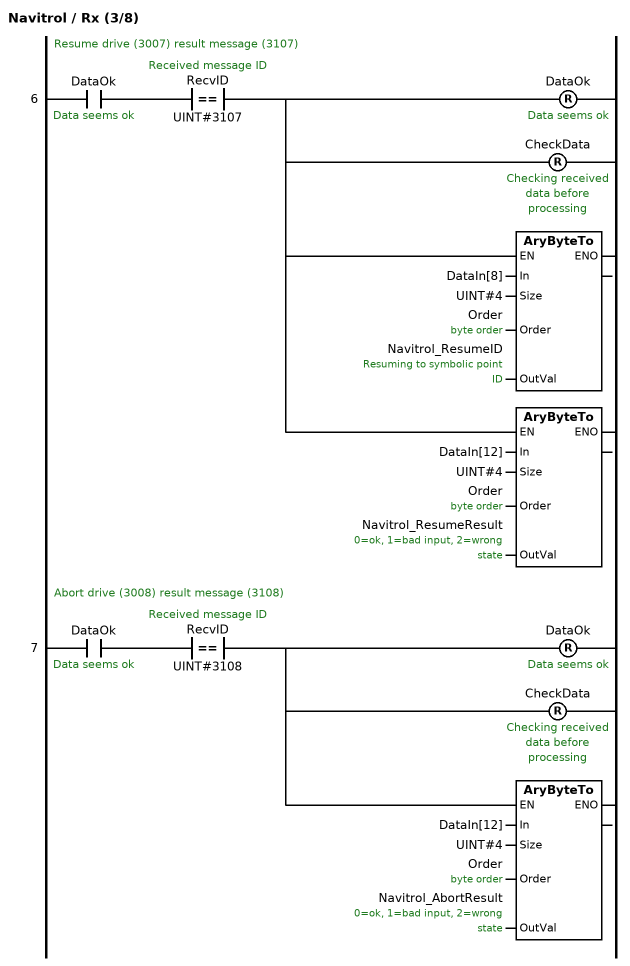
(* Rung 6: Resume drive (3007) result message (3107) *)
_p10 := DataOk AND (RecvID = UINT#3107);
IF _p10 THEN
    DataOk := FALSE;
    CheckData := FALSE;
    AryByteTo(In := DataIn[8], Size := UINT#4, Order := Order, OutVal := Navitrol_ResumeID);
    AryByteTo(In := DataIn[12], Size := UINT#4, Order := Order, OutVal := Navitrol_ResumeResult);
END_IF;
(* Rung 7: Abort drive (3008) result message (3108) *)
_p11 := DataOk AND (RecvID = UINT#3108);
IF _p11 THEN
    DataOk := FALSE;
    CheckData := FALSE;
    AryByteTo(In := DataIn[12], Size := UINT#4, Order := Order, OutVal := Navitrol_AbortResult);
END_IF;

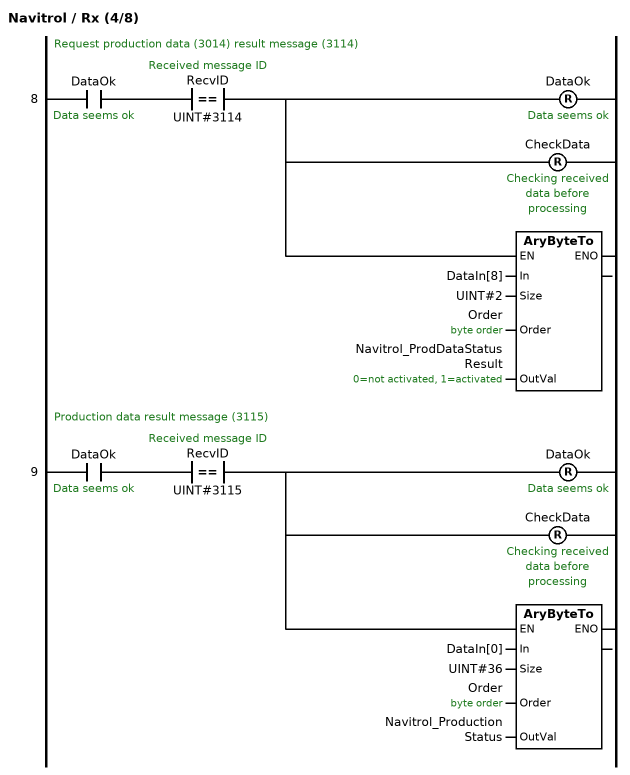
(* Rung 8: Request production data (3014) result message (3114) *)
_p12 := DataOk AND (RecvID = UINT#3114);
IF _p12 THEN
    DataOk := FALSE;
    CheckData := FALSE;
    AryByteTo(In := DataIn[8], Size := UINT#2, Order := Order, OutVal := Navitrol_ProdDataStatusResult);
END_IF;
(* Rung 9: Production data result message (3115) *)
_p13 := DataOk AND (RecvID = UINT#3115);
IF _p13 THEN
    DataOk := FALSE;
    CheckData := FALSE;
    AryByteTo(In := DataIn[0], Size := UINT#36, Order := Order, OutVal := Navitrol_ProductionStatus);
END_IF;

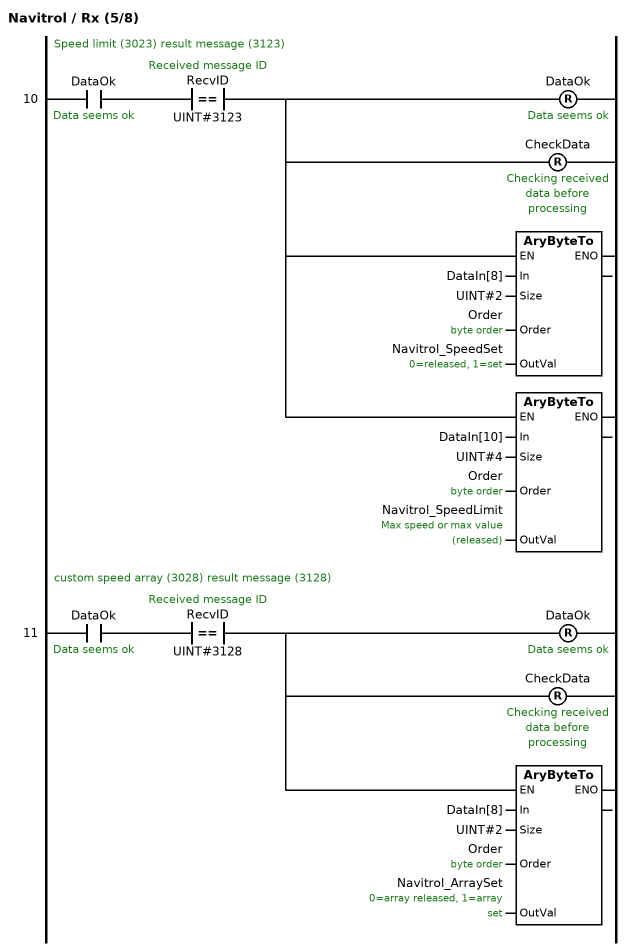
(* Rung 10: Speed limit (3023) result message (3123) *)
_p14 := DataOk AND (RecvID = UINT#3123);
IF _p14 THEN
    DataOk := FALSE;
    CheckData := FALSE;
    AryByteTo(In := DataIn[8], Size := UINT#2, Order := Order, OutVal := Navitrol_SpeedSet);
    AryByteTo(In := DataIn[10], Size := UINT#4, Order := Order, OutVal := Navitrol_SpeedLimit);
END_IF;
(* Rung 11: custom speed array (3028) result message (3128) *)
_p15 := DataOk AND (RecvID = UINT#3128);
IF _p15 THEN
    DataOk := FALSE;
    CheckData := FALSE;
    AryByteTo(In := DataIn[8], Size := UINT#2, Order := Order, OutVal := Navitrol_ArraySet);
END_IF;

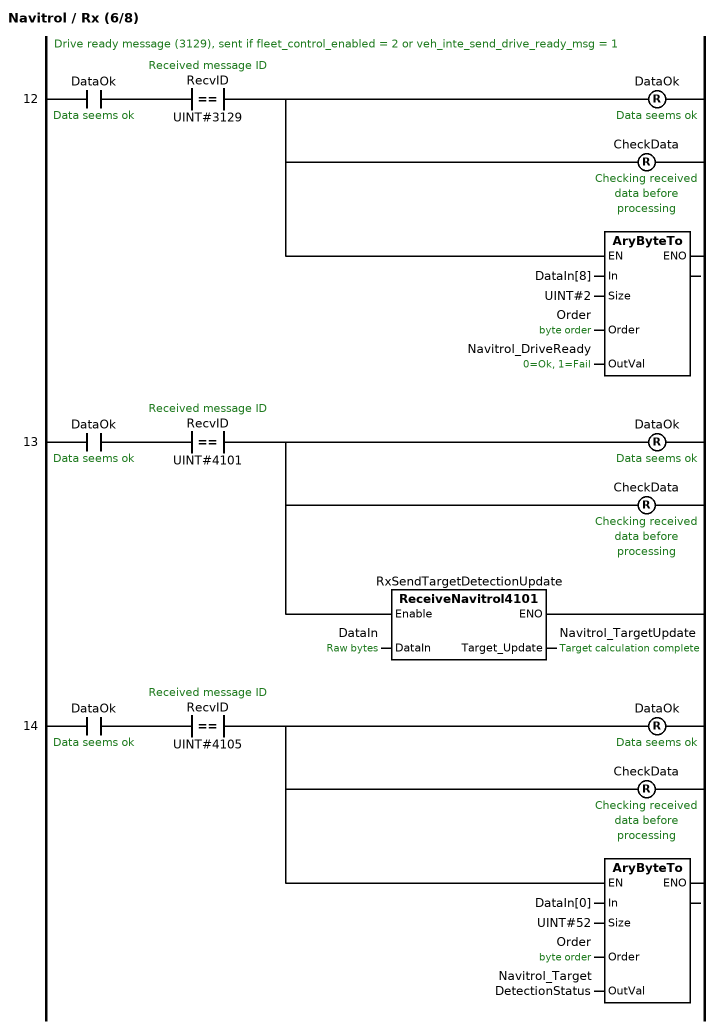
(* Rung 12: Drive ready message (3129), sent if fleet_control_enabled = 2 or veh_inte_send_drive_ready_msg = 1 *)
_p16 := DataOk AND (RecvID = UINT#3129);
IF _p16 THEN
    DataOk := FALSE;
    CheckData := FALSE;
    AryByteTo(In := DataIn[8], Size := UINT#2, Order := Order, OutVal := Navitrol_DriveReady);
END_IF;
(* Rung 13 *)
_p17 := DataOk AND (RecvID = UINT#4101);
IF _p17 THEN
    DataOk := FALSE;
    CheckData := FALSE;
END_IF;
RxSendTargetDetectionUpdate(Enable := _p17, DataIn := DataIn, Target_Update => Navitrol_TargetUpdate);
(* Rung 14 *)
_p18 := DataOk AND (RecvID = UINT#4105);
IF _p18 THEN
    DataOk := FALSE;
    CheckData := FALSE;
    AryByteTo(In := DataIn[0], Size := UINT#52, Order := Order, OutVal := Navitrol_TargetDetectionStatus);
END_IF;

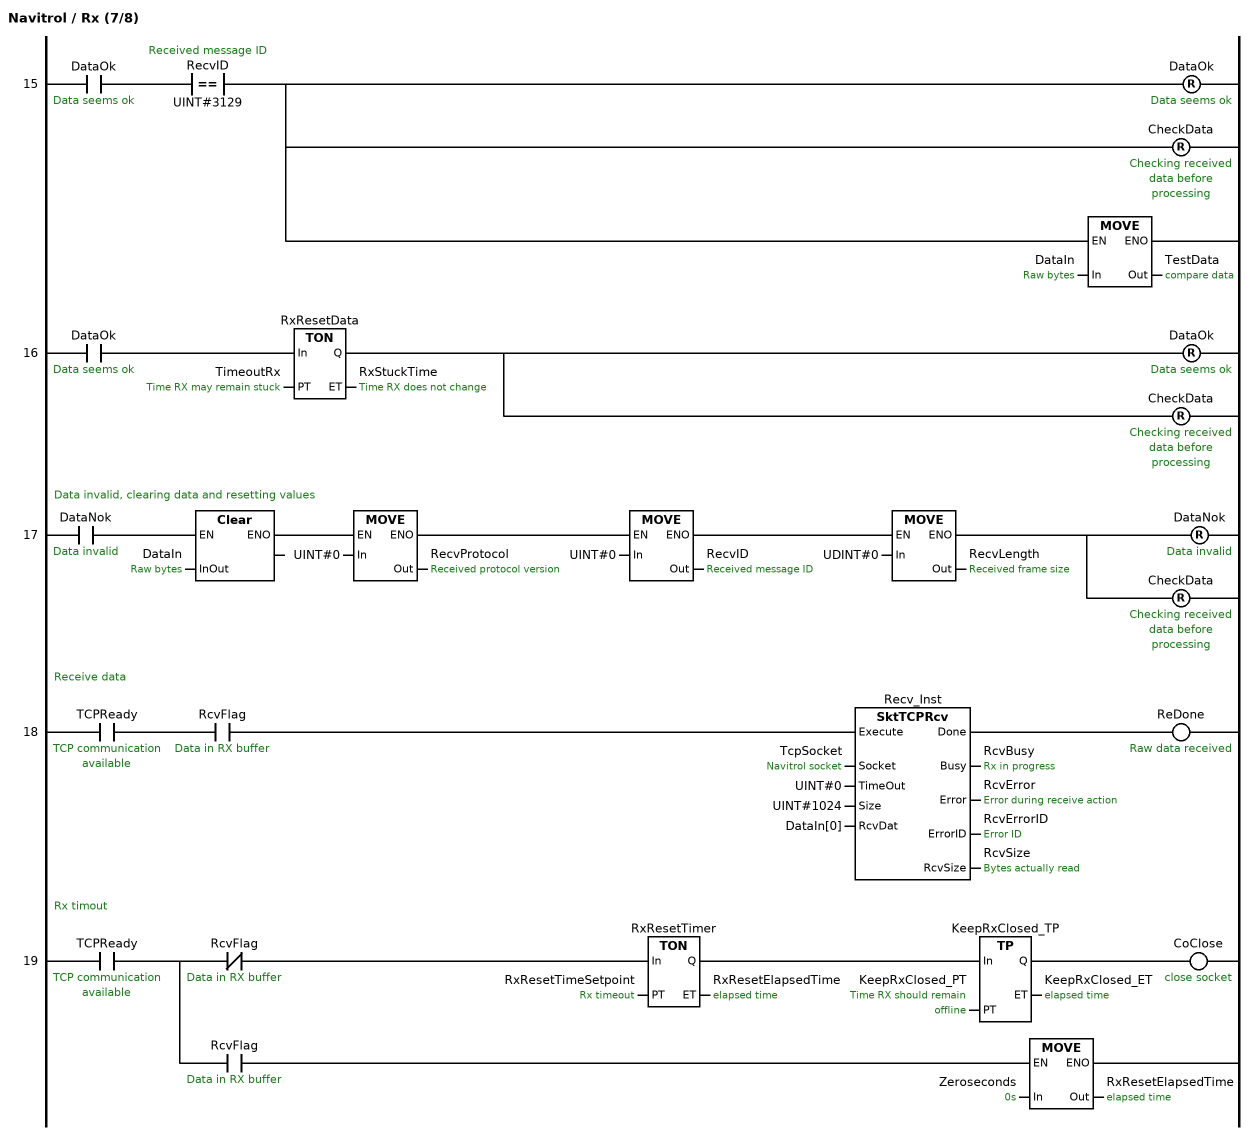
(* Rung 15 *)
_p19 := DataOk AND (RecvID = UINT#3129);
IF _p19 THEN
    DataOk := FALSE;
    CheckData := FALSE;
    TestData := DataIn;
END_IF;
(* Rung 16 *)
RxResetData(In := DataOk, PT := TimeoutRx, ET => RxStuckTime);
IF RxResetData.Q THEN
    DataOk := FALSE;
    CheckData := FALSE;
END_IF;
(* Rung 17: Data invalid, clearing data and resetting values *)
IF DataNok THEN
    Clear(InOut := DataIn);
    RecvProtocol := UINT#0;
    RecvID := UINT#0;
    RecvLength := UDINT#0;
END_IF;
_p20 := DataNok;
IF _p20 THEN
    DataNok := FALSE;
    CheckData := FALSE;
END_IF;
(* Rung 18: Receive data *)
Recv_Inst(Execute := TCPReady AND RcvFlag, Socket := TcpSocket, TimeOut := UINT#0, Size := UINT#1024, RcvDat := DataIn[0], Busy => RcvBusy, Error => RcvError, ErrorID => RcvErrorID, RcvSize => RcvSize);
ReDone := Recv_Inst.Done;
(* Rung 19: Rx timout *)
RxResetTimer(In := TCPReady AND NOT RcvFlag, PT := RxResetTimeSetpoint, ET => RxResetElapsedTime);
KeepRxClosed_TP(In := RxResetTimer.Q, PT := KeepRxClosed_PT, ET => KeepRxClosed_ET);
CoClose := KeepRxClosed_TP.Q;
IF TCPReady AND RcvFlag THEN RxResetElapsedTime := Zeroseconds; END_IF;

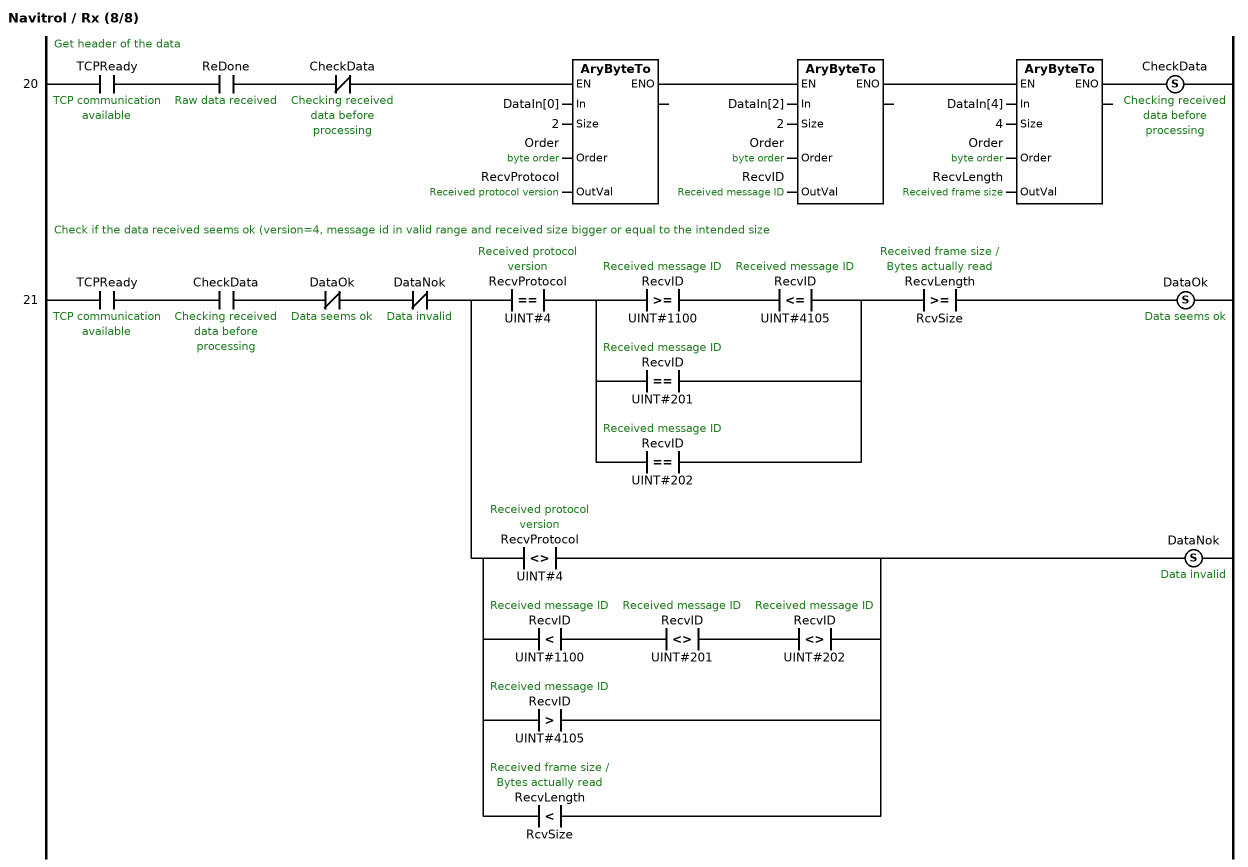
(* Rung 20: Get header of the data *)
IF TCPReady AND ReDone AND NOT CheckData THEN
    AryByteTo(In := DataIn[0], Size := 2, Order := Order, OutVal := RecvProtocol);
    AryByteTo(In := DataIn[2], Size := 2, Order := Order, OutVal := RecvID);
    AryByteTo(In := DataIn[4], Size := 4, Order := Order, OutVal := RecvLength);
    CheckData := TRUE;
END_IF;
(* Rung 21: Check if the data received seems ok (version=4, message id in valid range and received size bigger or equal to the intended size *)
_p21 := TCPReady AND CheckData AND NOT DataOk AND NOT DataNok;
IF _p21 AND (RecvProtocol = UINT#4) AND (((RecvID >= UINT#1100) AND (RecvID <= UINT#4105)) OR (RecvID = UINT#201) OR (RecvID = UINT#202)) AND (RecvLength >= RcvSize) THEN
    DataOk := TRUE;
END_IF;
IF _p21 AND ((RecvProtocol <> UINT#4) OR ((RecvID < UINT#1100) AND (RecvID <> UINT#201) AND (RecvID <> UINT#202)) OR (RecvID > UINT#4105) OR (RecvLength < RcvSize)) THEN
    DataNok := TRUE;
END_IF;
END_PROGRAM

PROGRAM IO_List
VAR
    Index : ULINT;
END_VAR
VAR_EXTERNAL
    Mqtt_values : ARRAY[0..32] OF MQTTval;
    HMI_Int3 : INT;
    HMI_Int2 : INT;
    HMI_Int6 : INT;
    AgvLoaded : BOOL;
    Estop_Out : BOOL;
    SafetyFieldNumber : INT;
    OptionalFieldReq : INT;
    HMI_Manual : BOOL;
    HMI_Input5 : BOOL;
    Brake_release : BOOL;
    HMI_Int10 : INT;
    ActuatorAction : BOOL;
    Scanner1_State : State_Scanner;
    Scanner3_State : State_Scanner;
    Scanner2_State : State_Scanner;
    LED_Reset : BOOL;
    Buzzer : BOOL;
    LED_Left : BOOL;
    LED_Right : BOOL;
    LED_Mid1 : BOOL;
    LED_Mid2 : BOOL;
    Lift_Control_Dir : BOOL;
    Indicator_Left : BOOL;
    Indicator_Right : BOOL;
    I00 : BOOL;
    I01 : BOOL;
    I02 : BOOL;
    I03 : BOOL;
    I04 : BOOL;
    Fork_bump_det_1 : BOOL;
    I05 : BOOL;
    Fork_bump_det_2 : BOOL;
    I06 : BOOL;
    Right_door_closed : BOOL;
    I07 : BOOL;
    Front_door_closed : BOOL;
    I08 : BOOL;
    Left_door_closed : BOOL;
    I09 : BOOL;
    Reset_Button : BOOL;
    I10 : BOOL;
    Brake_Override_Switch : BOOL;
    I11 : BOOL;
    Board_Detected : BOOL;
    I12 : BOOL;
    I13 : BOOL;
    O00 : BOOL;
    O01 : BOOL;
    O02 : BOOL;
    O03 : BOOL;
    O04 : BOOL;
    O05 : BOOL;
    O06 : BOOL;
    O07 : BOOL;
    O08 : BOOL;
    O09 : BOOL;
    N10_O00 : BOOL;
    N10_O01 : BOOL;
    N10_O02 : BOOL;
    Blue_spot1 : BOOL;
    Blue_spot2 : BOOL;
    Charge_Relay : BOOL;
    K11 : BOOL;
    N10_O03 : BOOL;
    N11_O00 : BOOL;
    K12 : BOOL;
    N11_O01 : BOOL;
    N11_O02 : BOOL;
    N11_O03 : BOOL;
    MES_State : Node_State;
    MES_Request_Cancel : BOOL;
    Estop_Channel1 : BOOL;
    SafetyStopped : BOOL;
    Error_Fork_Object : BOOL;
    ClientConnected : BOOL;
    MES_Cancel_Confirm : BOOL;
    Pressure_Sensor_Load : BOOL;
    Scan1_Warn : BOOL;
    Scan1_Slow : BOOL;
    Scan3_Warn : BOOL;
    Scan3_slow : BOOL;
    PalletDetection_state : Pallet_Det_State;
    CountedPallets : INT;
    lift_heavyLoad : BOOL;
    Scan2_Warn : BOOL;
    Scan2_Slow : BOOL;
    N3_N3_Si02 : BOOL;
    Lift_Sensor_Max : BOOL;
    LowObstacleIO : BOOL;
    Aout_1 : INT;
    LED_B : INT;
    LED_R : INT;
    Aout_2 : INT;
    LED_G : INT;
    Aout_4 : INT;
    Aout_3 : INT;
    Lift_Prop_Speed : INT;
END_VAR
//NX1 PLC IO
//Inputs
Scan1_Slow						:= I00;		//Front right warning field
Scan1_Warn 						:= I01;		//Front right stop field	
Scan2_Slow						:= I02;		//Front left warning field
Scan2_Warn	 					:= I03;		//Front left stop field
Scan3_Slow						:= I04;		//Rear stop field
Scan3_Warn 						:= I05;		//Rear Waring field
Right_door_closed				:= I06;		//Cover is closed
Front_door_closed				:= I07;		//Cover is closed
Left_door_closed				:= I08;		//Cover is closed
Reset_Button						:= I09;		//Reset input button
Fork_bump_det_1			:= I10;		//Fork tip sensor
Fork_bump_det_2			:= I11;		//fork tip sensor
Board_Detected 				:= I12;		//Board detection			
Brake_Override_Switch	:= I13;		//Brake release 
			

//Outputs
O00      :=     LED_Reset; 				//Indicator light
O01      :=     Buzzer; 					//Audio output
O02		:=		LED_Left;					//Disable left LED bar
O03 		:=		LED_Right;				//Disable right LED bar
O04 		:=		LED_Mid1	;				//Disable middle-right LED bar
O05 		:=		LED_Mid2	;				//Disable middle-left LED
O06 		:=		Brake_release;			//Brakes manual release


//High power outputs on NX1 bus
N10_O00	:=	Blue_spot1;		//Front facing Bluespot
N10_O01	:=	Charge_Relay;	//Enable contact power	
N10_O02	:= K11; 					//K11 is Valve Lift down
N10_O03	:= K12 ;					//K12 is Valve Lift up

//ECC203 Ethercat module
// Safety inputs 
Lift_Sensor_Max				:=	N3_N3_Si02;		// Lift hight max

Aout_1 := LED_R;
Aout_2 := LED_G;
Aout_3 := LED_B;
Aout_4 := Lift_Prop_Speed;
END_PROGRAM

FUNCTION_BLOCK PWM
VAR
    out : BOOL;  (* Enable output *)
    TOF_pulse : TOF;
    Period : BOOL;
    TOF_period : TOF;
    Period_ET : TIME;  (* elaped time *)
    Pulse_ET : TIME;  (* elapsed time *)
END_VAR
VAR_INPUT
    In : BOOL;  (* Enable *)
    Sync : BOOL;  (* Pulse to reset *)
    TimePeriod : TIME;  (* Time per cycle *)
    TimePulse : TIME;  (* Time on *)
END_VAR
VAR
    _e1 : F_TRIG;
END_VAR
(* ladder, written here as Structured Text *)

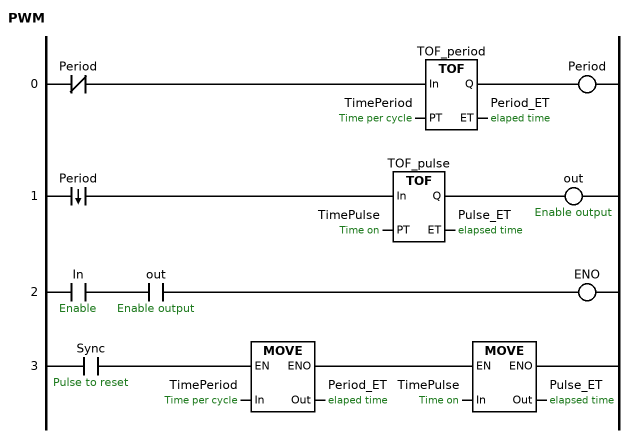
(* Rung 0 *)
TOF_period(In := NOT Period, PT := TimePeriod, ET => Period_ET);
Period := TOF_period.Q;
(* Rung 1 *)
_e1(CLK := Period);
TOF_pulse(In := _e1.Q, PT := TimePulse, ET => Pulse_ET);
out := TOF_pulse.Q;
(* Rung 2 *)
ENO := In AND out;
(* Rung 3 *)
IF Sync THEN
    Period_ET := TimePeriod;
    Pulse_ET := TimePulse;
END_IF;
END_FUNCTION_BLOCK

FUNCTION_BLOCK Ramp
VAR
    Target_Old : INT;
    Time_Ratio : REAL;
    TP_Ramp : TP;
END_VAR
VAR_INPUT
    In : BOOL;
    Target : INT;
    Period : TIME;
END_VAR
VAR_OUTPUT
    Out : INT;
END_VAR
VAR_INPUT
    Offset : INT := 0;  (* Optional *)
END_VAR
VAR
    _e1 : R_TRIG;
    _e2 : F_TRIG;
END_VAR
(* ladder, written here as Structured Text *)

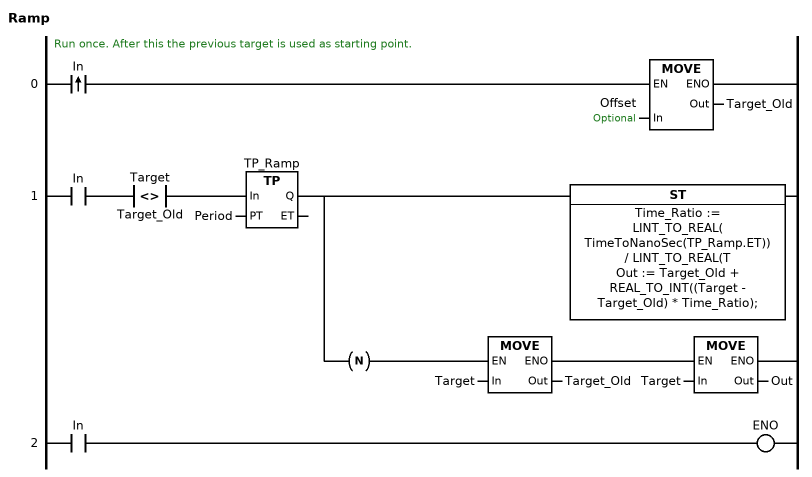
(* Rung 0: Run once. After this the previous target is used as starting point. *)
_e1(CLK := In);
IF _e1.Q THEN Target_Old := Offset; END_IF;
(* Rung 1 *)
TP_Ramp(In := In AND (Target <> Target_Old), PT := Period);
IF TP_Ramp.Q THEN
    Time_Ratio := LINT_TO_REAL(TimeToNanoSec(TP_Ramp.ET)) / LINT_TO_REAL(TimeToNanoSec(Period));
    Out := Target_Old + REAL_TO_INT((Target - Target_Old) * Time_Ratio);
END_IF;
_e2(CLK := TP_Ramp.Q);
IF _e2.Q THEN
    Target_Old := Target;
    Out := Target;
END_IF;
(* Rung 2 *)
ENO := In;
END_FUNCTION_BLOCK

FUNCTION_BLOCK Damp
VAR
    potition_ratio : REAL;
    position_start : INT;
    position_start_set : BOOL := False;
    setpoint_start_set : INT;
END_VAR
VAR_INPUT
    In : BOOL;
    position_current : INT;
    position_end : INT;
    setpoint_start : INT;
    setpoint_end : INT;
END_VAR
VAR_OUTPUT
    setpoint_current : INT;
END_VAR
IF In THEN
	IF NOT position_start_set THEN
		setpoint_start_set := setpoint_start;
		position_start := position_current;
		position_start_set := TRUE;
	END_IF;
	potition_ratio := INT_TO_REAL(position_end - position_current) / INT_TO_REAL(position_end - position_start);
	potition_ratio := ABS(potition_ratio);
	setpoint_current := setpoint_end + REAL_TO_INT((setpoint_start_set - setpoint_end) * potition_ratio);
ELSE
	position_start_set := FALSE;
	setpoint_current := 0;
END_IF;

ENO := In;
END_FUNCTION_BLOCK

FUNCTION_BLOCK GetToken
VAR
    Value : UINT;
    Begin_Value : UINT;
    ASCII : ARRAY[0..9] OF BYTE := [16#30, 16#31, 16#32, 16#33, 16#34, 16#35, 16#36, 16#37, 16#38, 16#39];
    Index1 : INT;
    Index2 : INT;
    Index3 : INT;
    Index4 : INT;
    Index5 : INT;
END_VAR
VAR_INPUT
    Convert : BOOL;
    WebToken : UINT;
END_VAR
VAR_OUTPUT
    Token1 : BYTE;
    Token2 : BYTE;
    Token3 : BYTE;
    Token4 : BYTE;
    Token5 : BYTE;
END_VAR
IF Convert THEN
	IF WebToken <> 0 THEN
		Begin_Value := WebToken;										//save start value
		Index1 := UINT_TO_INT(Begin_Value / 10000);		//How often is 10K in the value
		Value := Begin_Value - (10000 * INT_TO_UINT(Index1));	//Reduce value with calcluated amount
		Token1 := ASCII[Index1];											//Convert to ascii
		
		Index2 := UINT_TO_INT(Value / 1000);					//How often is 1K in the remainder?
		Value := Value - (1000 * INT_TO_UINT(Index2));		//Reduce value with the calculated amount
		Token2 := ASCII[Index2];											//Convert to ascii
		
		Index3 := UINT_TO_INT(Value / 100);						//How often is 100 in the remainder?
		Value := Value - (100 * INT_TO_UINT(Index3));		//Reduce value with the calculated amount
		Token3 := ASCII[Index3];											//Convert to ascii
		
		Index4 :=UINT_TO_INT( Value / 10);						//How often is 10 in the remainder?
		Value := Value - (10 * INT_TO_UINT(Index4));			//Reduce the value with the calculated amount
		Token4 := ASCII[index4];											//Convert to ascii
		//last value cannot be more than 9
		Token5 :=ASCII[Value];												//Convert to ascii
	ELSE
		//base value is 00000
		Token1 := ASCII[0];
		Token2 := ASCII[0];
		Token3 := ASCII[0];
		Token4 := ASCII[0];
		Token5 := ASCII[0];
	END_IF;
	ENO := 1;
ELSE
	ENO := 0;
END_IF;
END_FUNCTION_BLOCK

FUNCTION_BLOCK SendSaveLog
VAR
    DataReady : BOOL;  (* Data set ready for transmission *)
    TxBusy : BOOL;  (* Transmission in progress *)
    Data : Navitrol_SaveLogs_struct;
    SendDat : ARRAY[0..7] OF BYTE;  (* Data to send *)
    Messagesize : UINT;  (* Amount of bytes *)
    SendData : SktTCPSend;
END_VAR
VAR_INPUT
    Enable : BOOL;  (* Request to send *)
END_VAR
VAR_OUTPUT
    Done : BOOL;  (* Transmission done *)
END_VAR
VAR_INPUT
    Socket : _sSOCKET;  (* Navitrol socket *)
END_VAR
VAR_OUTPUT
    Error : BOOL;  (* Error during transmission *)
    ErrorID : WORD;  (* Error ID *)
END_VAR
VAR
    _e1 : R_TRIG;
    _p2 : BOOL;
    _p3 : BOOL;
    _e4 : R_TRIG;
END_VAR
(* ladder, written here as Structured Text *)

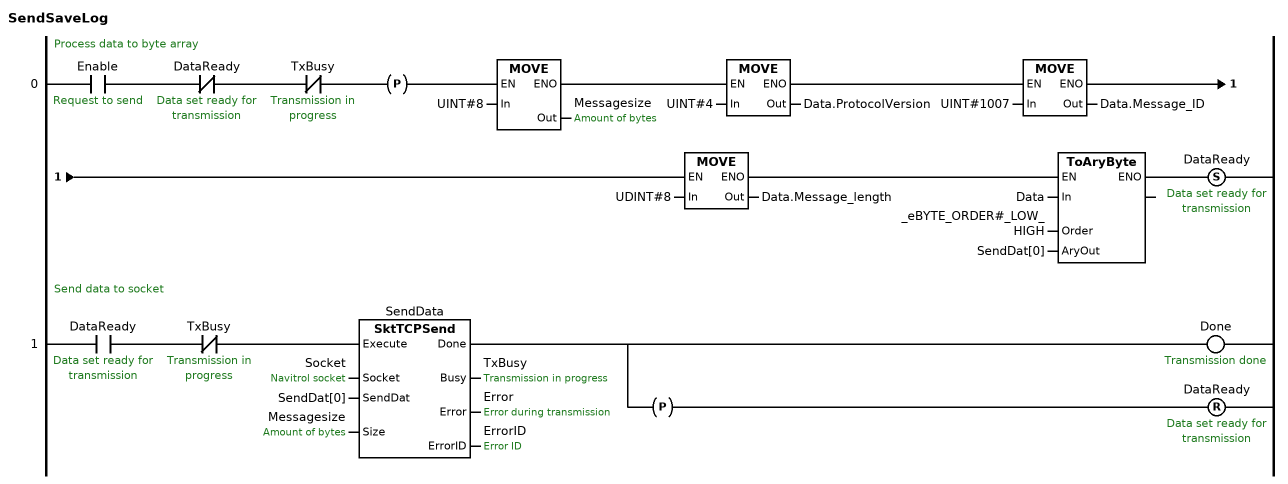
(* Rung 0: Process data to byte array *)
_e1(CLK := Enable AND NOT DataReady AND NOT TxBusy);
IF _e1.Q THEN
    Messagesize := UINT#8;
    Data.ProtocolVersion := UINT#4;
    Data.Message_ID := UINT#1007;
    Data.Message_length := UDINT#8;
    ToAryByte(In := Data, Order := _eBYTE_ORDER#_LOW_HIGH, AryOut := SendDat[0]);
    DataReady := TRUE;
END_IF;
(* Rung 1: Send data to socket *)
_p2 := DataReady AND NOT TxBusy;
SendData(Execute := _p2, Socket := Socket, SendDat := SendDat[0], Size := Messagesize, Busy => TxBusy, Error => Error, ErrorID => ErrorID);
_p3 := SendData.Done;
Done := _p3;
_e4(CLK := _p3);
IF _e4.Q THEN DataReady := FALSE; END_IF;
END_FUNCTION_BLOCK

FUNCTION_BLOCK SendPauseDrive
VAR
    DataReady : BOOL;  (* Data set ready for transmission *)
    TxBusy : BOOL;  (* Transmission in progress *)
    Data : Navitrol_PauseDrive_struct;
    SendDat : ARRAY[0..7] OF BYTE;  (* Data to send *)
    Messagesize : UINT;  (* Amount of bytes *)
    SendData : SktTCPSend;
END_VAR
VAR_INPUT
    Enable : BOOL;  (* Request to send *)
END_VAR
VAR_OUTPUT
    Done : BOOL;  (* Transmission done *)
END_VAR
VAR_INPUT
    Socket : _sSOCKET;  (* Navitrol socket *)
END_VAR
VAR_OUTPUT
    Error : BOOL;  (* Error during transmission *)
    ErrorID : WORD;  (* Error ID *)
END_VAR
VAR
    _e1 : R_TRIG;
    _p2 : BOOL;
    _p3 : BOOL;
    _e4 : R_TRIG;
END_VAR
(* ladder, written here as Structured Text *)

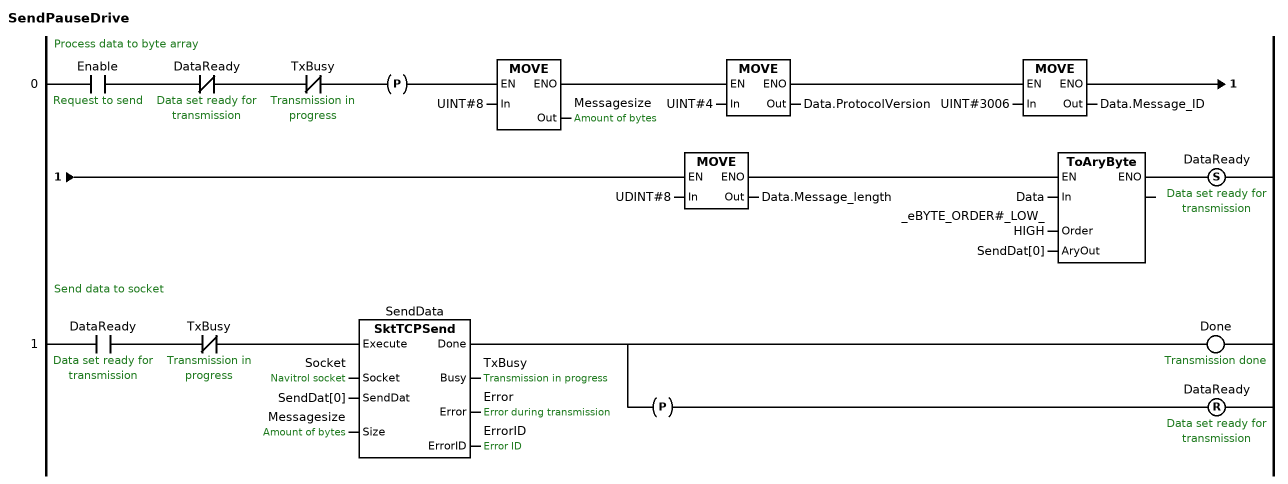
(* Rung 0: Process data to byte array *)
_e1(CLK := Enable AND NOT DataReady AND NOT TxBusy);
IF _e1.Q THEN
    Messagesize := UINT#8;
    Data.ProtocolVersion := UINT#4;
    Data.Message_ID := UINT#3006;
    Data.Message_length := UDINT#8;
    ToAryByte(In := Data, Order := _eBYTE_ORDER#_LOW_HIGH, AryOut := SendDat[0]);
    DataReady := TRUE;
END_IF;
(* Rung 1: Send data to socket *)
_p2 := DataReady AND NOT TxBusy;
SendData(Execute := _p2, Socket := Socket, SendDat := SendDat[0], Size := Messagesize, Busy => TxBusy, Error => Error, ErrorID => ErrorID);
_p3 := SendData.Done;
Done := _p3;
_e4(CLK := _p3);
IF _e4.Q THEN DataReady := FALSE; END_IF;
END_FUNCTION_BLOCK

FUNCTION_BLOCK SendResumeDrive
VAR
    DataReady : BOOL;  (* Data set ready for transmission *)
    TxBusy : BOOL;  (* Transmission in progress *)
    Data : Navitrol_ResumeDrive_struct;
    SendDat : ARRAY[0..7] OF BYTE;  (* Data to send *)
    Messagesize : UINT;  (* Amount of bytes *)
    SendData : SktTCPSend;
END_VAR
VAR_INPUT
    Enable : BOOL;  (* Request to send *)
END_VAR
VAR_OUTPUT
    Done : BOOL;  (* Transmission done *)
END_VAR
VAR_INPUT
    Socket : _sSOCKET;  (* Navitrol socket *)
END_VAR
VAR_OUTPUT
    Error : BOOL;  (* Error during transmission *)
    ErrorID : WORD;  (* Error ID *)
END_VAR
VAR
    _e1 : R_TRIG;
    _p2 : BOOL;
    _p3 : BOOL;
    _e4 : R_TRIG;
END_VAR
(* ladder, written here as Structured Text *)

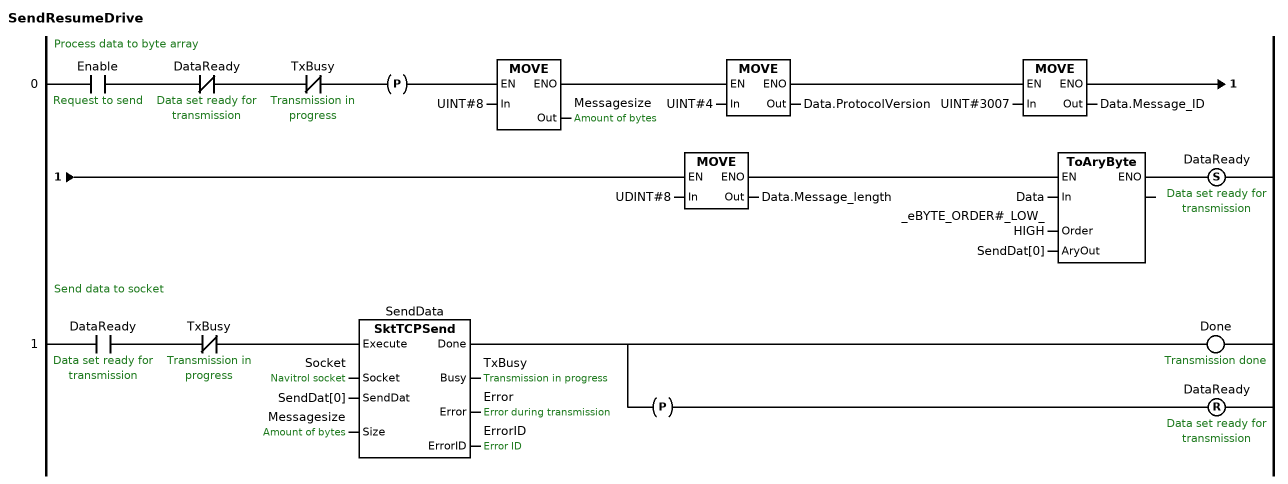
(* Rung 0: Process data to byte array *)
_e1(CLK := Enable AND NOT DataReady AND NOT TxBusy);
IF _e1.Q THEN
    Messagesize := UINT#8;
    Data.ProtocolVersion := UINT#4;
    Data.Message_ID := UINT#3007;
    Data.Message_length := UDINT#8;
    ToAryByte(In := Data, Order := _eBYTE_ORDER#_LOW_HIGH, AryOut := SendDat[0]);
    DataReady := TRUE;
END_IF;
(* Rung 1: Send data to socket *)
_p2 := DataReady AND NOT TxBusy;
SendData(Execute := _p2, Socket := Socket, SendDat := SendDat[0], Size := Messagesize, Busy => TxBusy, Error => Error, ErrorID => ErrorID);
_p3 := SendData.Done;
Done := _p3;
_e4(CLK := _p3);
IF _e4.Q THEN DataReady := FALSE; END_IF;
END_FUNCTION_BLOCK

FUNCTION_BLOCK SendAbortDrive
VAR
    DataReady : BOOL;  (* Data set ready for transmission *)
    TxBusy : BOOL;  (* Transmission in progress *)
    Data : Navitrol_AbortDrive_struct;
    SendDat : ARRAY[0..7] OF BYTE;  (* Data to send *)
    Messagesize : UINT;  (* Amount of bytes *)
    SendData : SktTCPSend;
END_VAR
VAR_INPUT
    Enable : BOOL;  (* Request to send *)
END_VAR
VAR_OUTPUT
    Done : BOOL;  (* Transmission done *)
END_VAR
VAR_INPUT
    Socket : _sSOCKET;  (* Navitrol socket *)
END_VAR
VAR_OUTPUT
    Error : BOOL;  (* Error during transmission *)
    ErrorID : WORD;  (* Error ID *)
END_VAR
VAR
    _e1 : R_TRIG;
    _p2 : BOOL;
    _p3 : BOOL;
    _e4 : R_TRIG;
END_VAR
(* ladder, written here as Structured Text *)

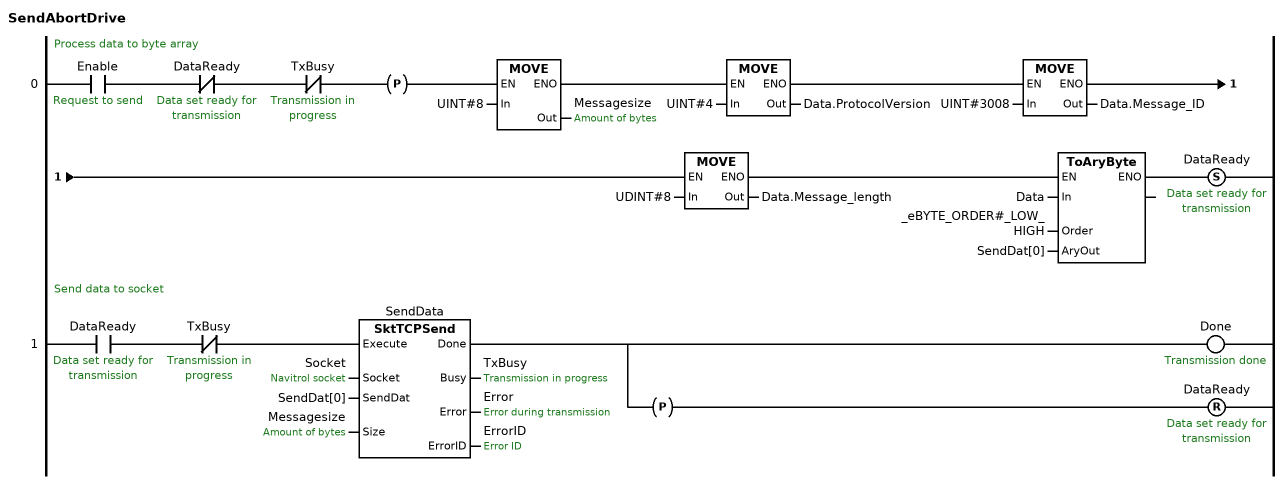
(* Rung 0: Process data to byte array *)
_e1(CLK := Enable AND NOT DataReady AND NOT TxBusy);
IF _e1.Q THEN
    Messagesize := UINT#8;
    Data.ProtocolVersion := UINT#4;
    Data.Message_ID := UINT#3008;
    Data.Message_length := UDINT#8;
    ToAryByte(In := Data, Order := _eBYTE_ORDER#_LOW_HIGH, AryOut := SendDat[0]);
    DataReady := TRUE;
END_IF;
(* Rung 1: Send data to socket *)
_p2 := DataReady AND NOT TxBusy;
SendData(Execute := _p2, Socket := Socket, SendDat := SendDat[0], Size := Messagesize, Busy => TxBusy, Error => Error, ErrorID => ErrorID);
_p3 := SendData.Done;
Done := _p3;
_e4(CLK := _p3);
IF _e4.Q THEN DataReady := FALSE; END_IF;
END_FUNCTION_BLOCK

FUNCTION_BLOCK SendSetSpeedLimit
VAR
    DataReady : BOOL;  (* data set ready for transmission *)
    TxBusy : BOOL;  (* Transmission in progress *)
    SendDat : ARRAY[0..13] OF BYTE;  (* Data to send *)
    Messagesize : UINT;  (* Amount of bytes *)
    Data : Navitrol_SetSpeedLimit_struct;  (* Message *)
    SendData : SktTCPSend;
    TimeoutTON : TON;
    Timeout_PT : TIME := 150ms;  (* Time until block can be re-enabled *)
    Timeout_ET : TIME;  (* elapsed time *)
    Timeout : BOOL;  (* Block time exceeded *)
END_VAR
VAR_INPUT
    Enable : BOOL;  (* Request to send *)
    Socket : _sSOCKET;  (* Navitrol socket *)
    SetRelease : BOOL;  (* False=use parameter values *)
    Speed : REAL;  (* Speed in m/s *)
END_VAR
VAR_OUTPUT
    Done : BOOL;  (* Transmission done *)
    Busy : BOOL;  (* Transmission in progress *)
    Error : BOOL;  (* Error during transmission *)
    ErrorID : WORD;  (* Error ID *)
END_VAR
VAR
    _p1 : BOOL;
    _p2 : BOOL;
    _e3 : R_TRIG;
END_VAR
(* ladder, written here as Structured Text *)

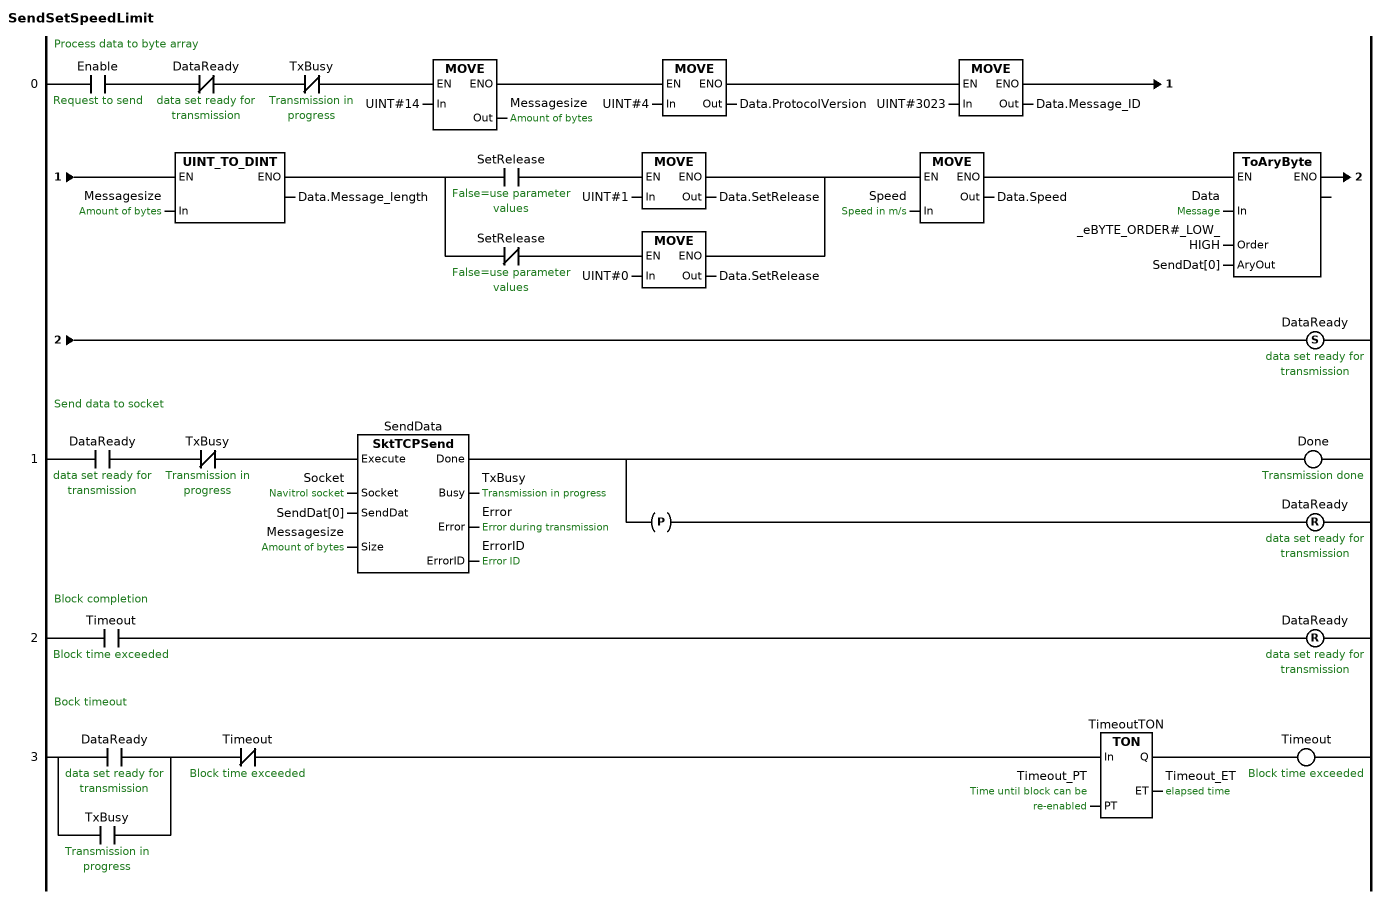
(* Rung 0: Process data to byte array *)
IF Enable AND NOT DataReady AND NOT TxBusy THEN
    Messagesize := UINT#14;
    Data.ProtocolVersion := UINT#4;
    Data.Message_ID := UINT#3023;
    Data.Message_length := UINT_TO_DINT(In := Messagesize);
END_IF;
IF Enable AND NOT DataReady AND NOT TxBusy AND SetRelease THEN Data.SetRelease := UINT#1; END_IF;
IF Enable AND NOT DataReady AND NOT TxBusy AND NOT SetRelease THEN Data.SetRelease := UINT#0; END_IF;
IF Enable AND NOT DataReady AND NOT TxBusy AND (SetRelease OR NOT SetRelease) THEN
    Data.Speed := Speed;
    ToAryByte(In := Data, Order := _eBYTE_ORDER#_LOW_HIGH, AryOut := SendDat[0]);
    DataReady := TRUE;
END_IF;
(* Rung 1: Send data to socket *)
_p1 := DataReady AND NOT TxBusy;
SendData(Execute := _p1, Socket := Socket, SendDat := SendDat[0], Size := Messagesize, Busy => TxBusy, Error => Error, ErrorID => ErrorID);
_p2 := SendData.Done;
Done := _p2;
_e3(CLK := _p2);
IF _e3.Q THEN DataReady := FALSE; END_IF;
(* Rung 2: Block completion *)
IF Timeout THEN DataReady := FALSE; END_IF;
(* Rung 3: Bock timeout *)
TimeoutTON(In := (DataReady OR TxBusy) AND NOT Timeout, PT := Timeout_PT, ET => Timeout_ET);
Timeout := TimeoutTON.Q;
END_FUNCTION_BLOCK

FUNCTION_BLOCK SendSetTargetDetectionMode
VAR
    DataReady : BOOL;  (* data set ready for transmission *)
    Messagesize : UINT;  (* Amount of bytes *)
    SendDat : ARRAY[0..47] OF BYTE;  (* Data to send *)
    SendData : SktTCPSend;
    TxBusy : BOOL;  (* Transmission in progress *)
END_VAR
VAR_OUTPUT
    Done : BOOL;  (* Transmission done *)
    Busy : BOOL;  (* Transmission in progress *)
    Error : BOOL;  (* Error during transmission *)
    ErrorID : WORD;  (* Error ID *)
END_VAR
VAR_INPUT
    Enable : BOOL;  (* Request to send *)
    Socket : _sSOCKET;  (* Navitrol socket *)
    Data : Navitrol_SetTargetDetectionControlModeLift_struct;  (* Target detection settings *)
END_VAR
VAR
    _e1 : R_TRIG;
    _p2 : BOOL;
    _p3 : BOOL;
    _e4 : R_TRIG;
END_VAR
(* ladder, written here as Structured Text *)

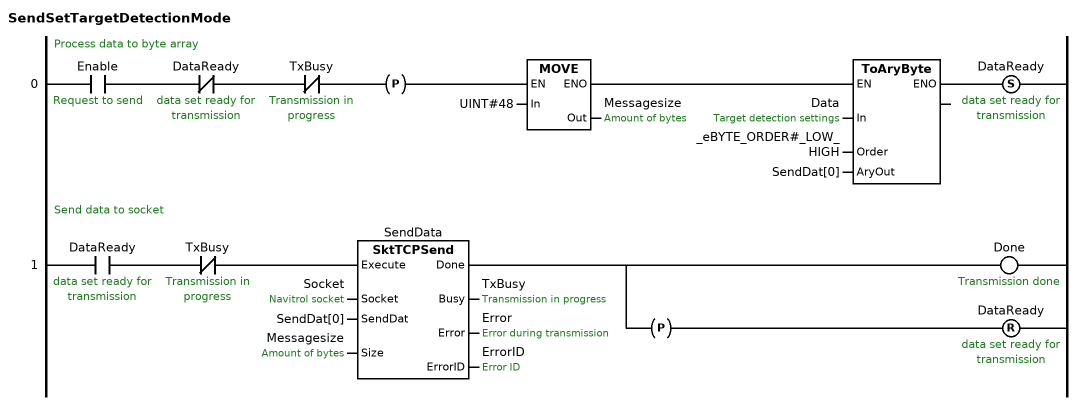
(* Rung 0: Process data to byte array *)
_e1(CLK := Enable AND NOT DataReady AND NOT TxBusy);
IF _e1.Q THEN
    Messagesize := UINT#48;
    ToAryByte(In := Data, Order := _eBYTE_ORDER#_LOW_HIGH, AryOut := SendDat[0]);
    DataReady := TRUE;
END_IF;
(* Rung 1: Send data to socket *)
_p2 := DataReady AND NOT TxBusy;
SendData(Execute := _p2, Socket := Socket, SendDat := SendDat[0], Size := Messagesize, Busy => TxBusy, Error => Error, ErrorID => ErrorID);
_p3 := SendData.Done;
Done := _p3;
_e4(CLK := _p3);
IF _e4.Q THEN DataReady := FALSE; END_IF;
END_FUNCTION_BLOCK

FUNCTION_BLOCK SendAbortWithData
VAR
    DataReady : BOOL;  (* Data set ready for transmission *)
    TxBusy : BOOL;  (* Transmission in progress *)
    Data : Navitrol_AbortWithData_struct;
    SendDat : ARRAY[0..13] OF BYTE;  (* Data to send *)
    Messagesize : UINT;  (* Amount of bytes *)
    SendData : SktTCPSend;
END_VAR
VAR_INPUT
    Enable : BOOL;  (* Request to send *)
END_VAR
VAR_OUTPUT
    Done : BOOL;  (* Transmission done *)
END_VAR
VAR_INPUT
    Socket : _sSOCKET;  (* Navitrol socket *)
    Completed : BOOL;  (* Drive is done *)
END_VAR
VAR_OUTPUT
    Error : BOOL;  (* Error during transmission *)
    ErrorID : WORD;  (* Error ID *)
END_VAR
VAR
    _e1 : R_TRIG;
    _p2 : BOOL;
    _p3 : BOOL;
    _e4 : R_TRIG;
END_VAR
(* ladder, written here as Structured Text *)

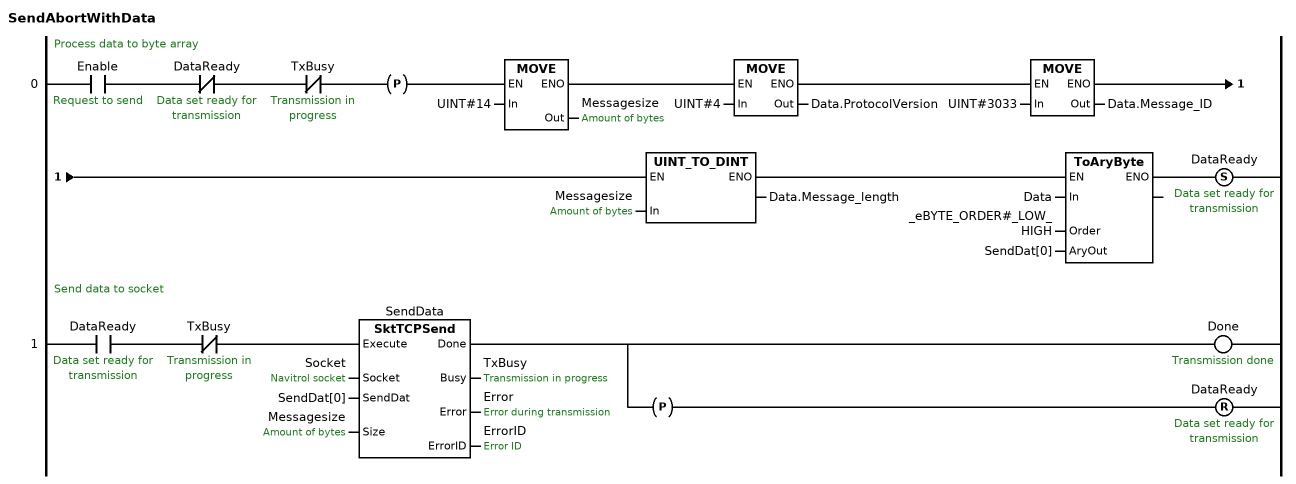
(* Rung 0: Process data to byte array *)
_e1(CLK := Enable AND NOT DataReady AND NOT TxBusy);
IF _e1.Q THEN
    Messagesize := UINT#14;
    Data.ProtocolVersion := UINT#4;
    Data.Message_ID := UINT#3033;
    Data.Message_length := UINT_TO_DINT(In := Messagesize);
    ToAryByte(In := Data, Order := _eBYTE_ORDER#_LOW_HIGH, AryOut := SendDat[0]);
    DataReady := TRUE;
END_IF;
(* Rung 1: Send data to socket *)
_p2 := DataReady AND NOT TxBusy;
SendData(Execute := _p2, Socket := Socket, SendDat := SendDat[0], Size := Messagesize, Busy => TxBusy, Error => Error, ErrorID => ErrorID);
_p3 := SendData.Done;
Done := _p3;
_e4(CLK := _p3);
IF _e4.Q THEN DataReady := FALSE; END_IF;
END_FUNCTION_BLOCK

FUNCTION_BLOCK SendRequestDriveReady
VAR
    DataReady : BOOL;  (* Data set ready for transmission *)
    TxBusy : BOOL;  (* Transmission in progress *)
    Messagesize : UINT;  (* Amount of bytes *)
    Data : Navitrol_RequestDriveCompleted_struct;  (* Message *)
    SendData : SktTCPSend;
    SendDat : ARRAY[0..13] OF BYTE;  (* Data to send *)
    Timeout_TON : TON;
    Max_Time : TIME := 150ms;  (* Timeout *)
    Timeout_ET : TIME;  (* elapsed time *)
END_VAR
VAR_INPUT
    Enable : BOOL;  (* Request to send *)
    Socket : _sSOCKET;  (* Navitrol socket *)
    ReadyType : UINT;  (* Request type *)
END_VAR
VAR_OUTPUT
    Done : BOOL;  (* Transmission done *)
    Busy : BOOL;  (* Transmission in progress *)
    Error : BOOL;  (* Error during transmission *)
    ErrorID : WORD;  (* Error ID *)
END_VAR
VAR
    _e1 : R_TRIG;
    _p2 : BOOL;
    _p3 : BOOL;
    _e4 : R_TRIG;
END_VAR
(* ladder, written here as Structured Text *)

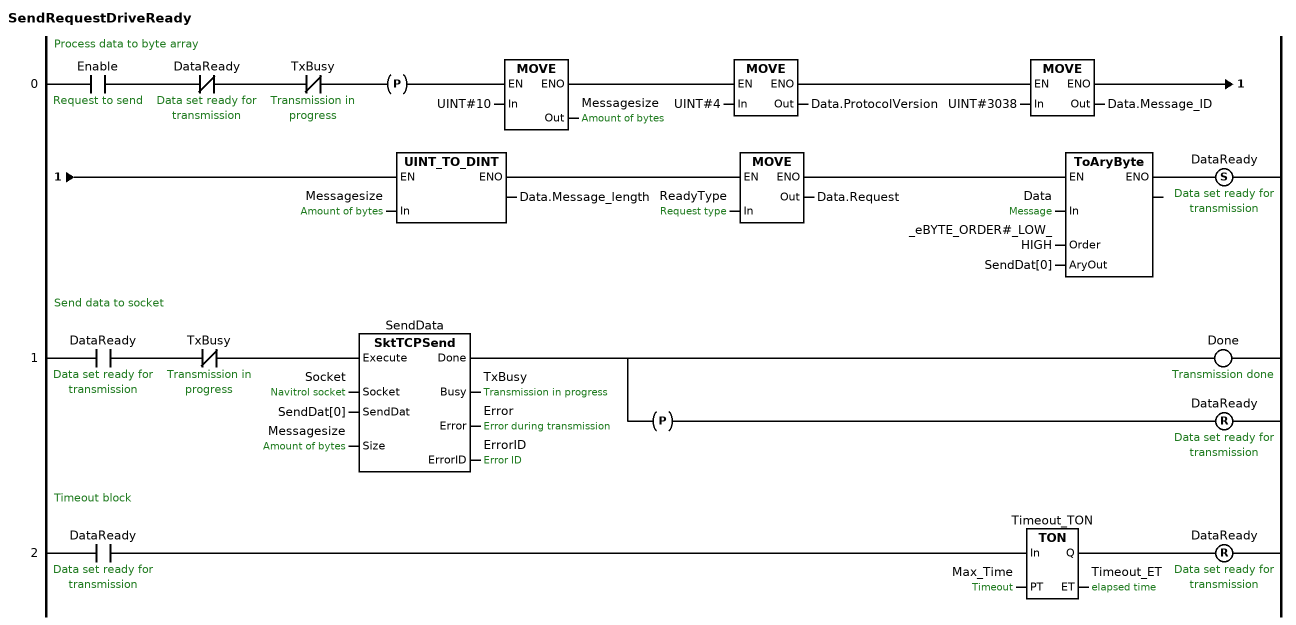
(* Rung 0: Process data to byte array *)
_e1(CLK := Enable AND NOT DataReady AND NOT TxBusy);
IF _e1.Q THEN
    Messagesize := UINT#10;
    Data.ProtocolVersion := UINT#4;
    Data.Message_ID := UINT#3038;
    Data.Message_length := UINT_TO_DINT(In := Messagesize);
    Data.Request := ReadyType;
    ToAryByte(In := Data, Order := _eBYTE_ORDER#_LOW_HIGH, AryOut := SendDat[0]);
    DataReady := TRUE;
END_IF;
(* Rung 1: Send data to socket *)
_p2 := DataReady AND NOT TxBusy;
SendData(Execute := _p2, Socket := Socket, SendDat := SendDat[0], Size := Messagesize, Busy => TxBusy, Error => Error, ErrorID => ErrorID);
_p3 := SendData.Done;
Done := _p3;
_e4(CLK := _p3);
IF _e4.Q THEN DataReady := FALSE; END_IF;
(* Rung 2: Timeout block *)
Timeout_TON(In := DataReady, PT := Max_Time, ET => Timeout_ET);
IF Timeout_TON.Q THEN DataReady := FALSE; END_IF;
END_FUNCTION_BLOCK

FUNCTION_BLOCK SendSetSpeedArray
VAR
    DataReady : BOOL;  (* data set ready for transmission *)
    TxBusy : BOOL;  (* Transmission in progress *)
    SendDat : ARRAY[0..11] OF BYTE;  (* Data to send *)
    Messagesize : UINT;  (* Amount of bytes *)
    Data : Navitrol_SetSpeedArray_struct;  (* Message *)
    SendData : SktTCPSend;
END_VAR
VAR_INPUT
    Enable : BOOL;  (* Request to send *)
    Socket : _sSOCKET;  (* Navitrol socket *)
    SetRelease : BOOL;  (* False=use parameter values *)
    ArrayIndex : UINT;  (* Array index 0..9 *)
END_VAR
VAR_OUTPUT
    Done : BOOL;  (* Transmission done *)
    Busy : BOOL;  (* Transmission in progress *)
    Error : BOOL;  (* Error during transmission *)
    ErrorID : WORD;  (* Error ID *)
END_VAR
VAR
    _e1 : R_TRIG;
    _p2 : BOOL;
    _p3 : BOOL;
    _e4 : R_TRIG;
END_VAR
(* ladder, written here as Structured Text *)

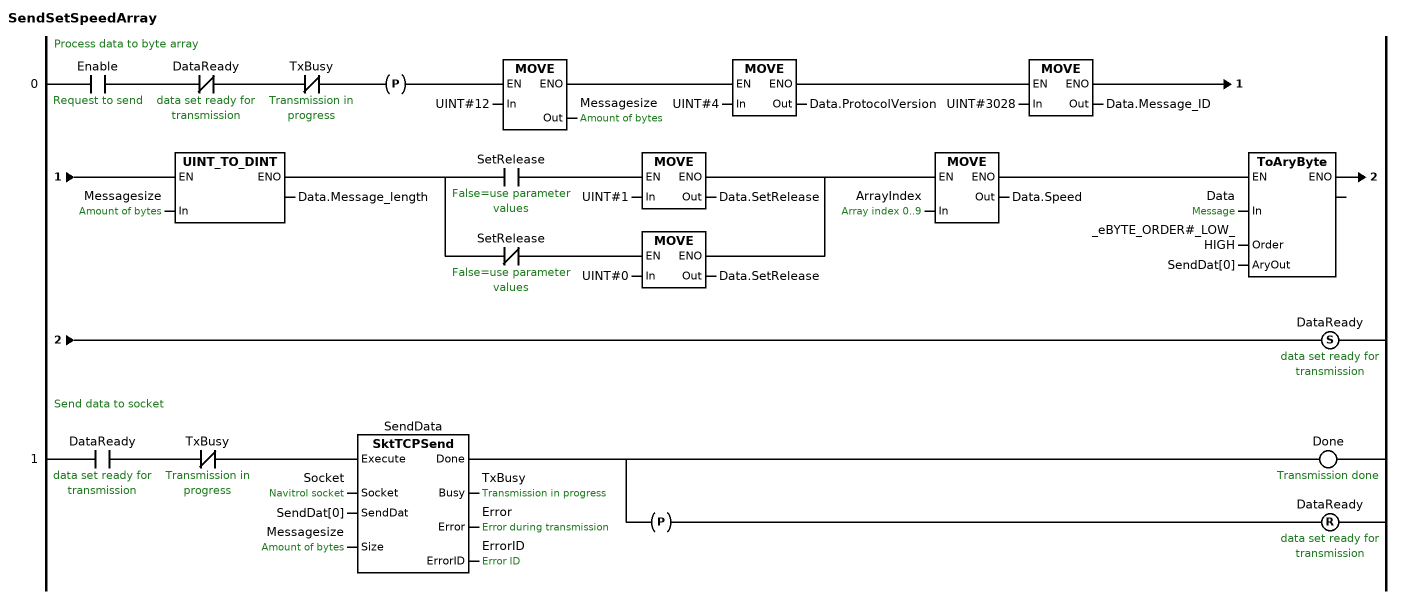
(* Rung 0: Process data to byte array *)
_e1(CLK := Enable AND NOT DataReady AND NOT TxBusy);
IF _e1.Q THEN
    Messagesize := UINT#12;
    Data.ProtocolVersion := UINT#4;
    Data.Message_ID := UINT#3028;
    Data.Message_length := UINT_TO_DINT(In := Messagesize);
END_IF;
IF _e1.Q AND SetRelease THEN Data.SetRelease := UINT#1; END_IF;
IF _e1.Q AND NOT SetRelease THEN Data.SetRelease := UINT#0; END_IF;
IF _e1.Q AND (SetRelease OR NOT SetRelease) THEN
    Data.Speed := ArrayIndex;
    ToAryByte(In := Data, Order := _eBYTE_ORDER#_LOW_HIGH, AryOut := SendDat[0]);
    DataReady := TRUE;
END_IF;
(* Rung 1: Send data to socket *)
_p2 := DataReady AND NOT TxBusy;
SendData(Execute := _p2, Socket := Socket, SendDat := SendDat[0], Size := Messagesize, Busy => TxBusy, Error => Error, ErrorID => ErrorID);
_p3 := SendData.Done;
Done := _p3;
_e4(CLK := _p3);
IF _e4.Q THEN DataReady := FALSE; END_IF;
END_FUNCTION_BLOCK

FUNCTION_BLOCK ReceiveNavitrol201
VAR
    Messagesize : UINT := 12;  (* Header size *)
    Order : _eBYTE_ORDER := _LOW_HIGH;  (* Byte order *)
    ErrorlistHeader : Navitrol_Errorlist_struct;
    Headerdone : BOOL;  (* Finished partial data *)
    counter : UDINT;  (* array index *)
    Datadone : BOOL;  (* Process completed *)
    Timeout_TON : TON;
    MaxTime : TIME := 100ms;  (* Max block time *)
    MaxTime_ET : TIME;  (* elapsed time *)
END_VAR
VAR_INPUT
    Enable : BOOL;
    DataIn : ARRAY[0..1023] OF BYTE;  (* Raw data *)
END_VAR
VAR_OUTPUT
    ErrorCount : UDINT;  (* Amount of errors received *)
    ErrorList : ARRAY[0..9] OF UDINT;  (* Error list (max 10) *)
END_VAR
VAR
    _e1 : R_TRIG;
    _e2 : R_TRIG;
END_VAR
(* ladder, written here as Structured Text *)

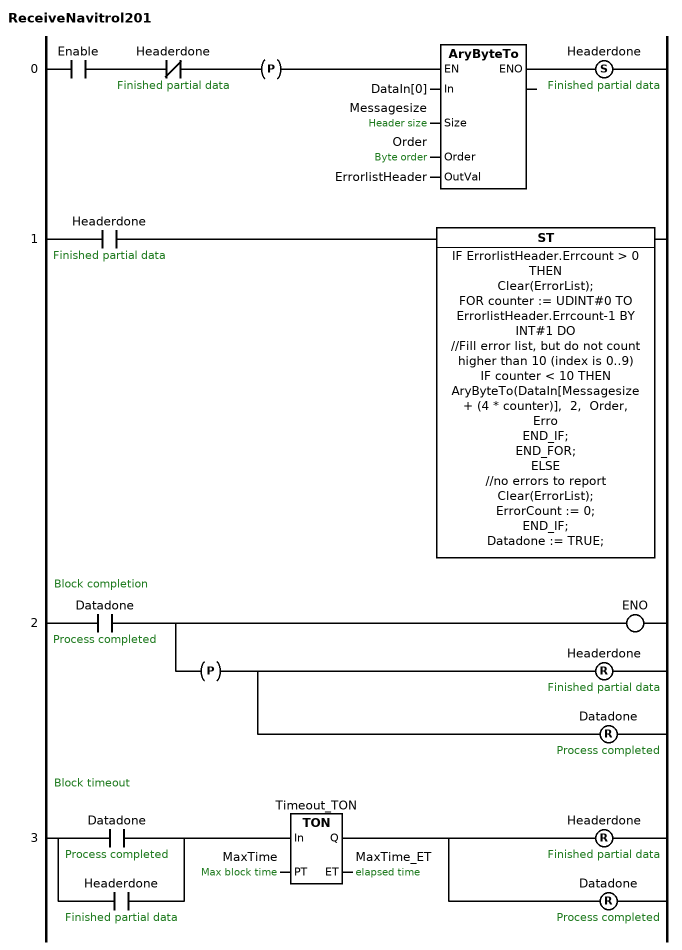
(* Rung 0 *)
_e1(CLK := Enable AND NOT Headerdone);
IF _e1.Q THEN
    AryByteTo(In := DataIn[0], Size := Messagesize, Order := Order, OutVal := ErrorlistHeader);
    Headerdone := TRUE;
END_IF;
(* Rung 1 *)
IF Headerdone THEN
    IF ErrorlistHeader.Errcount > 0 THEN
    	Clear(ErrorList);
    	FOR counter := UDINT#0 TO ErrorlistHeader.Errcount-1 BY INT#1 DO
    		//Fill error list, but do not count higher than 10 (index is 0..9)
    		IF counter < 10 THEN
    			AryByteTo(DataIn[Messagesize + (4 * counter)], 	2,	Order,	ErrorList[counter]);
    		END_IF;
    	END_FOR;
    ELSE
    	//no errors to report
    	Clear(ErrorList);
    	ErrorCount := 0;
    END_IF;
    
    Datadone := TRUE;
END_IF;
(* Rung 2: Block completion *)
ENO := Datadone;
_e2(CLK := Datadone);
IF _e2.Q THEN
    Headerdone := FALSE;
    Datadone := FALSE;
END_IF;
(* Rung 3: Block timeout *)
Timeout_TON(In := Datadone OR Headerdone, PT := MaxTime, ET => MaxTime_ET);
IF Timeout_TON.Q THEN
    Headerdone := FALSE;
    Datadone := FALSE;
END_IF;
END_FUNCTION_BLOCK

FUNCTION_BLOCK SendSupervisorStatusLocal
(* Navitrol status message v4. / API document: v2.41 / Created: 8-Dec-2020 *)
VAR
    SendData : SktTCPSend;
    DataReady : BOOL;  (* data set ready for transmission *)
    SendDat : ARRAY[0..1024] OF BYTE;  (* Data to send *)
    Messagesize : UINT;  (* Amount of bytes *)
    Order : _eBYTE_ORDER := _LOW_HIGH;  (* Byte order (little/big endian) *)
    Selection : USINT;  (* Section process selector *)
    TxBusy : BOOL;  (* Transmission in progress *)
    DataProcess : BOOL;  (* Data being processed *)
    TxOffset : UDINT;  (* Byte offset *)
    InputOffset : INT;  (* Byte offset for variable input section *)
    index : INT;  (* Loop index *)
    TimeoutTON : TON;
    Timeout_PT : TIME := 150ms;  (* Time until block can be re-enabled *)
    Timeout_ET : TIME;  (* elapsed time *)
    Timeout : BOOL;  (* Took too long *)
END_VAR
VAR_OUTPUT
    Done : BOOL;  (* Transmission done *)
    Busy : BOOL;  (* Transmission active *)
    Error : BOOL;  (* Tx error *)
    ErrorID : WORD;  (* Error code *)
END_VAR
VAR_INPUT
    Enable : BOOL;  (* Request to send *)
    Socket : _sSOCKET;  (* Navitrol socket *)
    Default_section : PLC_Status_Struct;  (* Status message *)
    Actuator_section : PLC_Act_Sec_Struct;  (* ID1 *)
    Manual_section : PLC_Navitrol_Manual_struct;  (* ID2 *)
    Error_section : PLC_Err_sec_struct;  (* ID3 *)
    Error_list : ARRAY[0..4] OF PLC_Error_struct;  (* ID3 *)
    Warning_list : ARRAY[0..4] OF PLC_Warn_struct;  (* ID3 *)
    Inputs_section : Navitrol_Status_inputs_struct;  (* ID4 *)
    Scanner_section : PLC_Navitrol_Status_laserscanner_struct;  (* ID5 *)
    Remote_section : PLC_Navitrol_Joystick_struct;  (* ID6 *)
    DriveCon_section : PLC_Navitrol_DriveControl_struct;  (* ID7 *)
    Battery_section : Navitrol_Status_Battery_struct;  (* ID8 *)
END_VAR
VAR_EXTERNAL
    NrOfSections : UINT;
    Sections : ARRAY[1..10] OF UINT;
END_VAR
VAR
    _e1 : R_TRIG;
    _p2 : BOOL;
    _e3 : R_TRIG;
    _p4 : BOOL;
    _e5 : R_TRIG;
    _p6 : BOOL;
    _e7 : R_TRIG;
    _e8 : R_TRIG;
    _e9 : R_TRIG;
    _p10 : BOOL;
    _e11 : R_TRIG;
    _p12 : BOOL;
    _e13 : R_TRIG;
    _p14 : BOOL;
    _e15 : R_TRIG;
    _p16 : BOOL;
    _e17 : R_TRIG;
    _p18 : BOOL;
    _p19 : BOOL;
    _e20 : R_TRIG;
END_VAR
(* ladder, written here as Structured Text *)

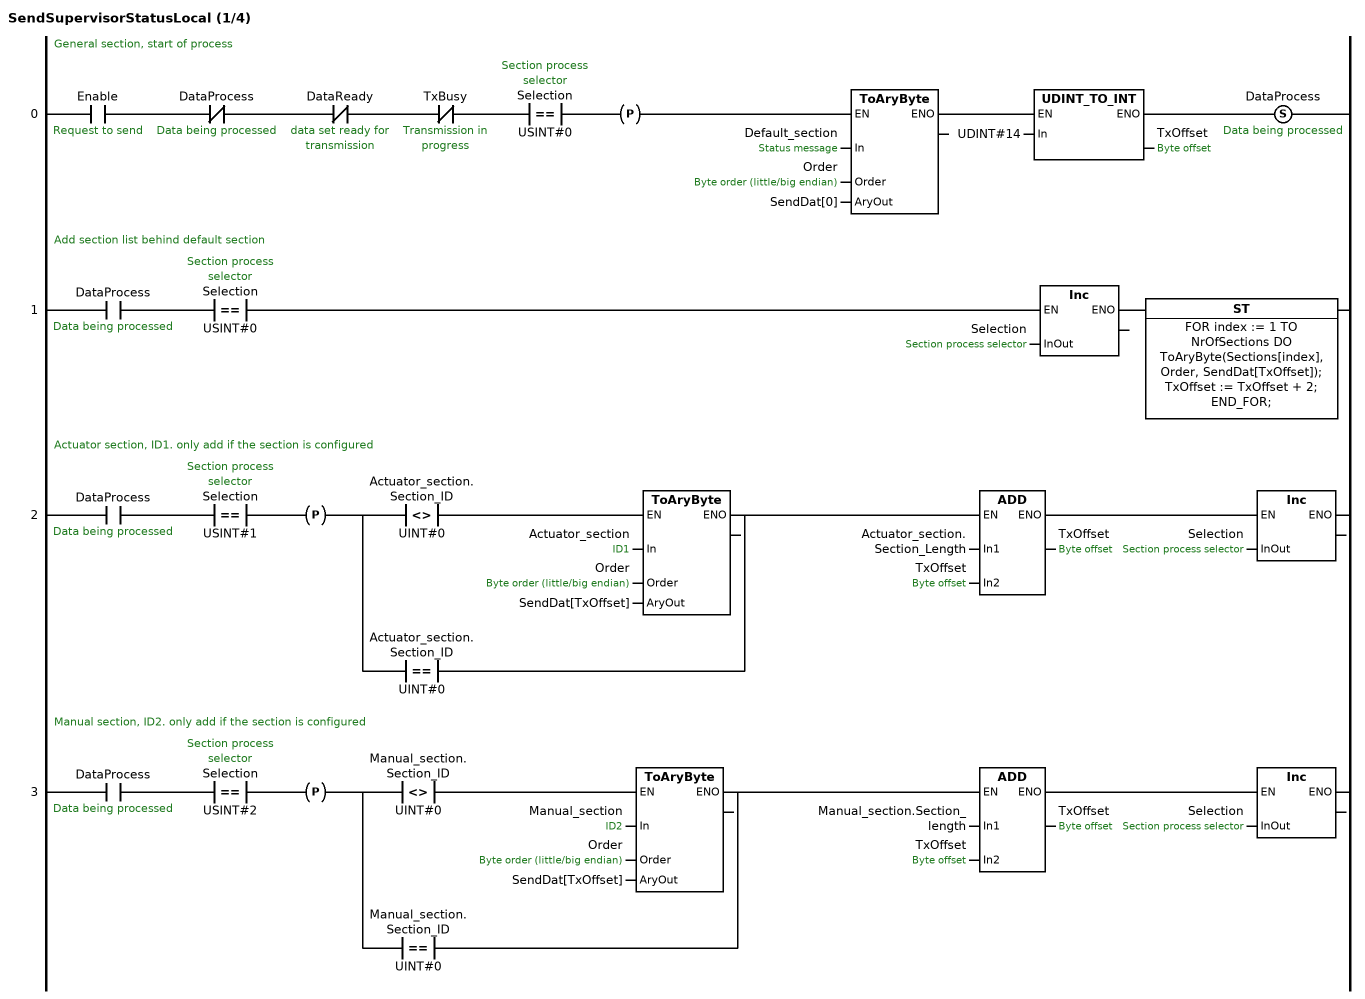
(* Rung 0: General section, start of process *)
_e1(CLK := Enable AND NOT DataProcess AND NOT DataReady AND NOT TxBusy AND (Selection = USINT#0));
IF _e1.Q THEN
    ToAryByte(In := Default_section, Order := Order, AryOut := SendDat[0]);
    TxOffset := UDINT_TO_INT(In := UDINT#14);
    DataProcess := TRUE;
END_IF;
(* Rung 1: Add section list behind default section *)
_p2 := DataProcess AND (Selection = USINT#0);
IF _p2 THEN Inc(InOut := Selection); END_IF;
IF _p2 THEN
    FOR index := 1 TO NrOfSections DO
    	ToAryByte(Sections[index], Order, SendDat[TxOffset]);
    	TxOffset := TxOffset + 2;
    END_FOR;
END_IF;
(* Rung 2: Actuator section, ID1. only add if the section is configured *)
_e3(CLK := DataProcess AND (Selection = USINT#1));
_p4 := _e3.Q AND (Actuator_section.Section_ID <> UINT#0);
IF _p4 THEN ToAryByte(In := Actuator_section, Order := Order, AryOut := SendDat[TxOffset]); END_IF;
IF _p4 OR (_e3.Q AND (Actuator_section.Section_ID = UINT#0)) THEN
    TxOffset := Actuator_section.Section_Length + TxOffset;
    Inc(InOut := Selection);
END_IF;
(* Rung 3: Manual section, ID2. only add if the section is configured *)
_e5(CLK := DataProcess AND (Selection = USINT#2));
_p6 := _e5.Q AND (Manual_section.Section_ID <> UINT#0);
IF _p6 THEN ToAryByte(In := Manual_section, Order := Order, AryOut := SendDat[TxOffset]); END_IF;
IF _p6 OR (_e5.Q AND (Manual_section.Section_ID = UINT#0)) THEN
    TxOffset := Manual_section.Section_length + TxOffset;
    Inc(InOut := Selection);
END_IF;

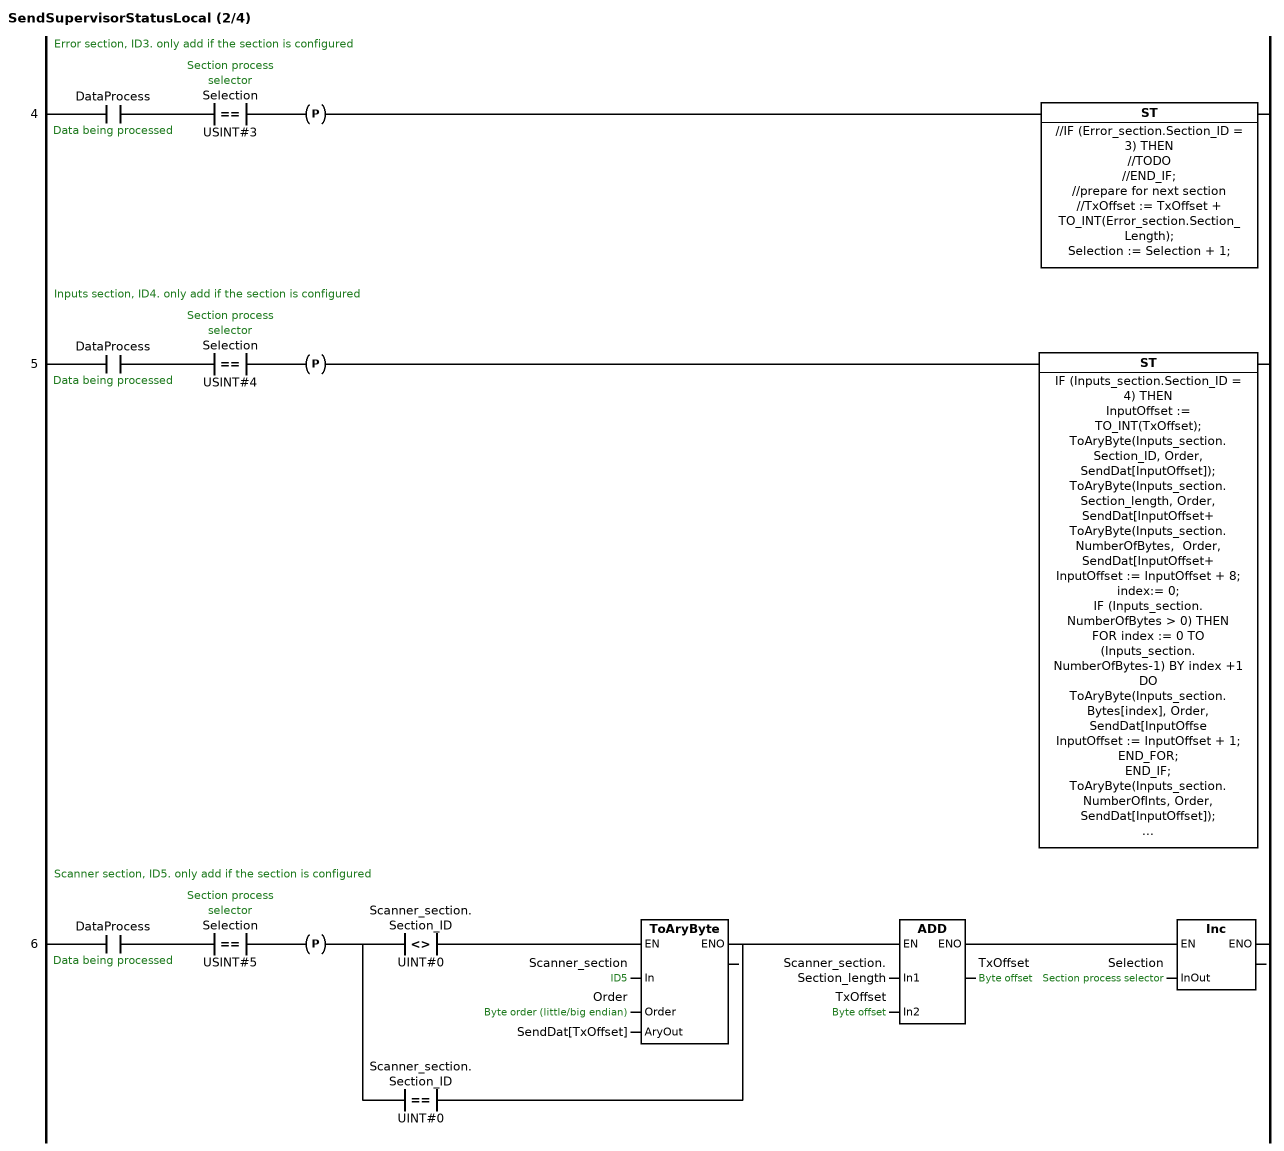
(* Rung 4: Error section, ID3. only add if the section is configured *)
_e7(CLK := DataProcess AND (Selection = USINT#3));
IF _e7.Q THEN
    //IF (Error_section.Section_ID = 3) THEN
    	//TODO
    //END_IF;
    
    //prepare for next section
    //TxOffset := TxOffset + TO_INT(Error_section.Section_Length);
    Selection := Selection + 1;
END_IF;
(* Rung 5: Inputs section, ID4. only add if the section is configured *)
_e8(CLK := DataProcess AND (Selection = USINT#4));
IF _e8.Q THEN
    IF (Inputs_section.Section_ID = 4) THEN
    	InputOffset := TO_INT(TxOffset);
    	ToAryByte(Inputs_section.Section_ID, Order, SendDat[InputOffset]);
    	ToAryByte(Inputs_section.Section_length, Order, SendDat[InputOffset+2]);
    	ToAryByte(Inputs_section.NumberOfBytes,	 Order, SendDat[InputOffset+6]);
    	InputOffset := InputOffset + 8;
    	index:= 0;
    	IF (Inputs_section.NumberOfBytes > 0) THEN
    		FOR index := 0 TO (Inputs_section.NumberOfBytes-1) BY index +1 DO
    			ToAryByte(Inputs_section.Bytes[index], Order, SendDat[InputOffset]);
    			InputOffset := InputOffset + 1;
    		END_FOR;
    	END_IF;
    	ToAryByte(Inputs_section.NumberOfInts, Order, SendDat[InputOffset]);
    	InputOffset := InputOffset + 2;
    	index:= 0;
    	IF (Inputs_section.NumberOfInts > 0) THEN
    		FOR index := 0 TO (Inputs_section.NumberOfInts-1) BY index +1 DO
    			ToAryByte(Inputs_section.Ints[index], Order, SendDat[InputOffset]);
    			InputOffset := InputOffset + 4;
    		END_FOR;
    	END_IF;
    	ToAryByte(Inputs_section.NumberOfFloats, Order, SendDat[InputOffset]);
    	InputOffset := InputOffset + 2;
    	index:= 0;
    	IF (Inputs_section.NumberOfFloats > 0) THEN
    		FOR index := 0 TO (Inputs_section.NumberOfFloats-1) BY index +1 DO
    			ToAryByte(Inputs_section.Floats[index], Order, SendDat[InputOffset]);
    			InputOffset := InputOffset + 4;
    		END_FOR;
    	END_IF;
    END_IF;
    
    //prepare for next section
    TxOffset := TxOffset + TO_INT(Inputs_section.Section_length);
    Selection := Selection + 1;
END_IF;
(* Rung 6: Scanner section, ID5. only add if the section is configured *)
_e9(CLK := DataProcess AND (Selection = USINT#5));
_p10 := _e9.Q AND (Scanner_section.Section_ID <> UINT#0);
IF _p10 THEN ToAryByte(In := Scanner_section, Order := Order, AryOut := SendDat[TxOffset]); END_IF;
IF _p10 OR (_e9.Q AND (Scanner_section.Section_ID = UINT#0)) THEN
    TxOffset := Scanner_section.Section_length + TxOffset;
    Inc(InOut := Selection);
END_IF;

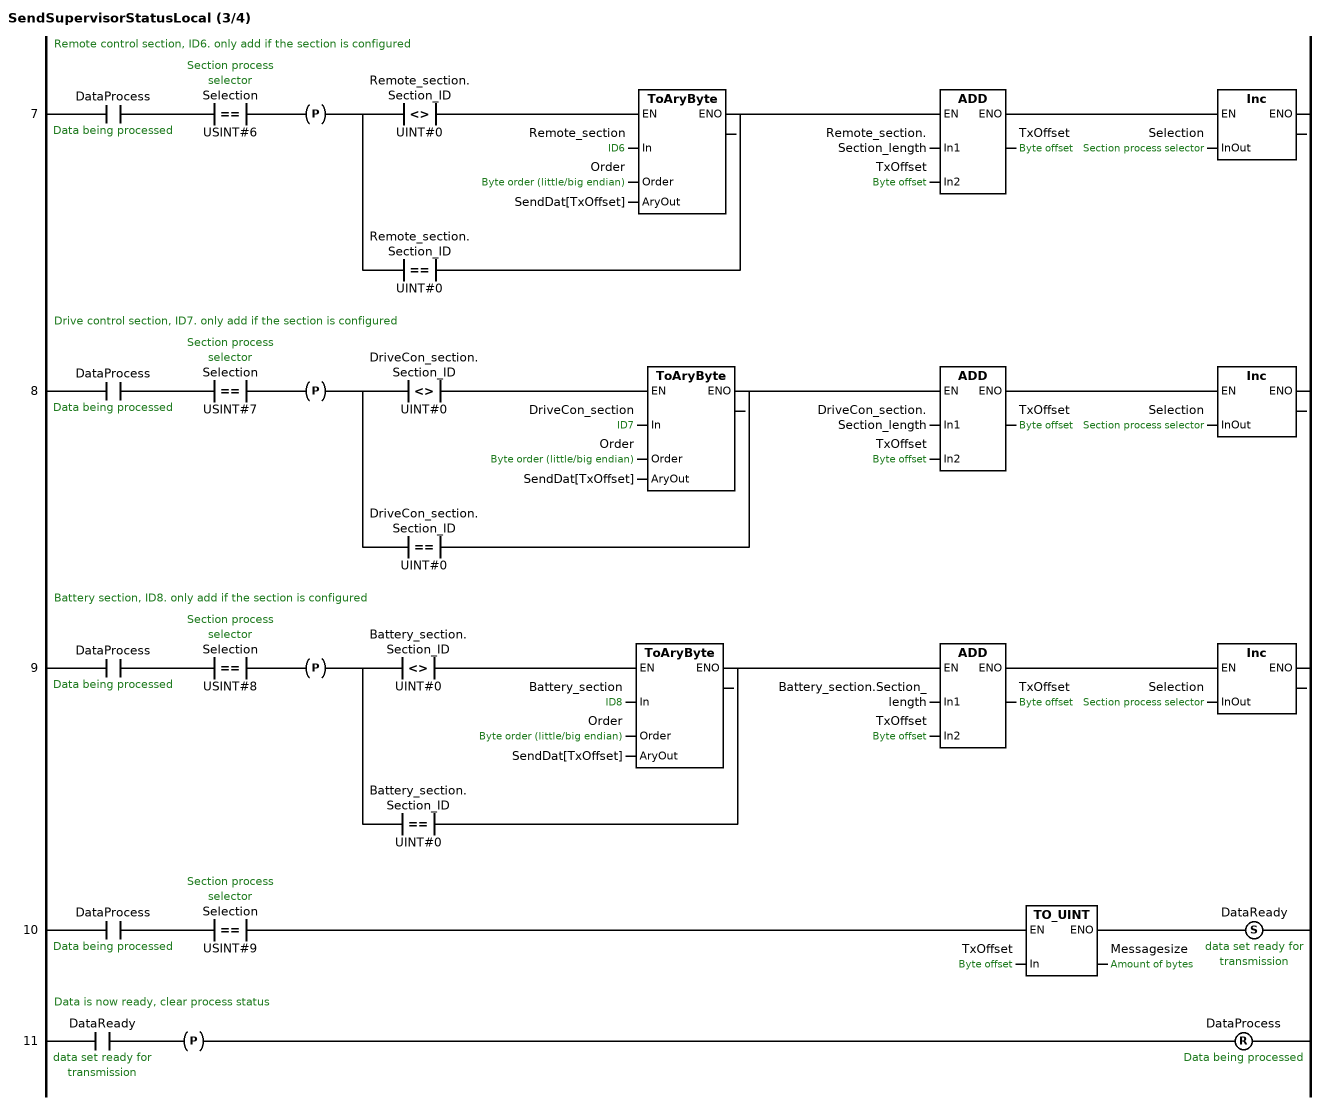
(* Rung 7: Remote control section, ID6. only add if the section is configured *)
_e11(CLK := DataProcess AND (Selection = USINT#6));
_p12 := _e11.Q AND (Remote_section.Section_ID <> UINT#0);
IF _p12 THEN ToAryByte(In := Remote_section, Order := Order, AryOut := SendDat[TxOffset]); END_IF;
IF _p12 OR (_e11.Q AND (Remote_section.Section_ID = UINT#0)) THEN
    TxOffset := Remote_section.Section_length + TxOffset;
    Inc(InOut := Selection);
END_IF;
(* Rung 8: Drive control section, ID7. only add if the section is configured *)
_e13(CLK := DataProcess AND (Selection = USINT#7));
_p14 := _e13.Q AND (DriveCon_section.Section_ID <> UINT#0);
IF _p14 THEN ToAryByte(In := DriveCon_section, Order := Order, AryOut := SendDat[TxOffset]); END_IF;
IF _p14 OR (_e13.Q AND (DriveCon_section.Section_ID = UINT#0)) THEN
    TxOffset := DriveCon_section.Section_length + TxOffset;
    Inc(InOut := Selection);
END_IF;
(* Rung 9: Battery section, ID8. only add if the section is configured *)
_e15(CLK := DataProcess AND (Selection = USINT#8));
_p16 := _e15.Q AND (Battery_section.Section_ID <> UINT#0);
IF _p16 THEN ToAryByte(In := Battery_section, Order := Order, AryOut := SendDat[TxOffset]); END_IF;
IF _p16 OR (_e15.Q AND (Battery_section.Section_ID = UINT#0)) THEN
    TxOffset := Battery_section.Section_length + TxOffset;
    Inc(InOut := Selection);
END_IF;
(* Rung 10 *)
IF DataProcess AND (Selection = USINT#9) THEN
    Messagesize := TO_UINT(In := TxOffset);
    DataReady := TRUE;
END_IF;
(* Rung 11: Data is now ready, clear process status *)
_e17(CLK := DataReady);
IF _e17.Q THEN DataProcess := FALSE; END_IF;

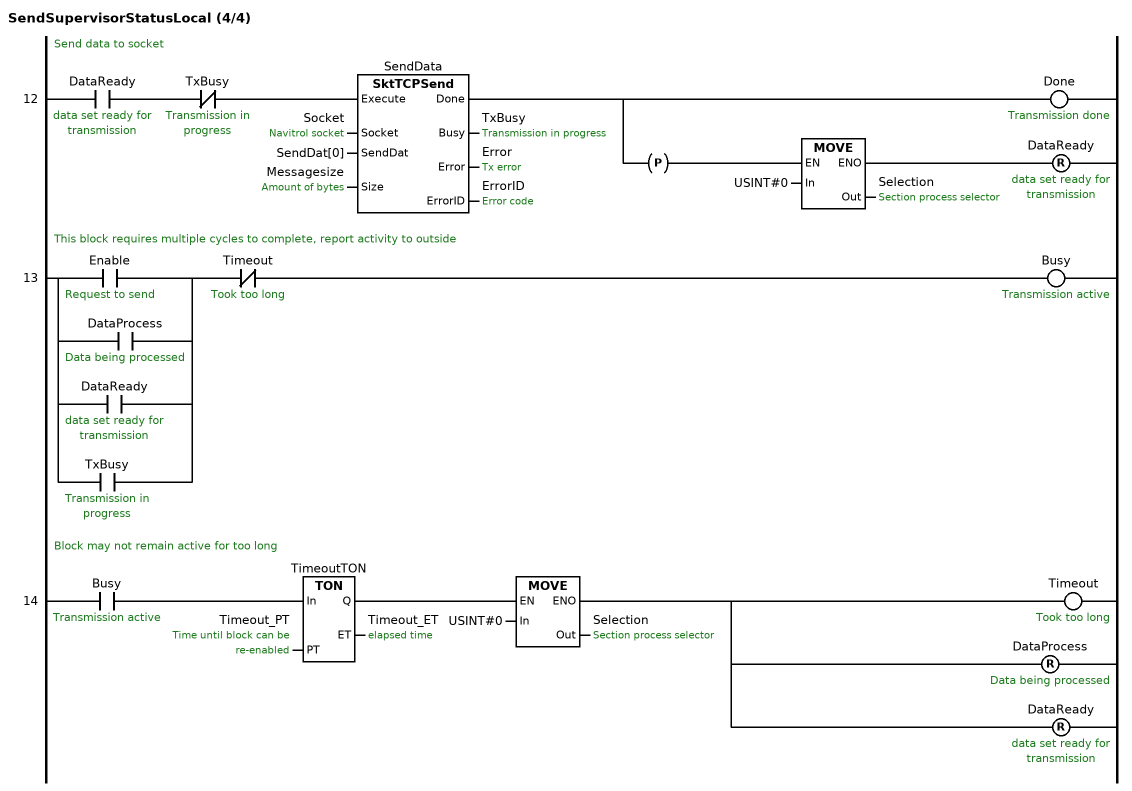
(* Rung 12: Send data to socket *)
_p18 := DataReady AND NOT TxBusy;
SendData(Execute := _p18, Socket := Socket, SendDat := SendDat[0], Size := Messagesize, Busy => TxBusy, Error => Error, ErrorID => ErrorID);
_p19 := SendData.Done;
Done := _p19;
_e20(CLK := _p19);
IF _e20.Q THEN
    Selection := USINT#0;
    DataReady := FALSE;
END_IF;
(* Rung 13: This block requires multiple cycles to complete, report activity to outside *)
Busy := (Enable OR DataProcess OR DataReady OR TxBusy) AND NOT Timeout;
(* Rung 14: Block may not remain active for too long *)
TimeoutTON(In := Busy, PT := Timeout_PT, ET => Timeout_ET);
IF TimeoutTON.Q THEN Selection := USINT#0; END_IF;
Timeout := TimeoutTON.Q;
IF TimeoutTON.Q THEN
    DataProcess := FALSE;
    DataReady := FALSE;
END_IF;
END_FUNCTION_BLOCK

FUNCTION_BLOCK SendRequestProductionStatus
VAR
    DataReady : BOOL;  (* Data set ready for transmission *)
    TxBusy : BOOL;  (* Transmission in progress *)
    Data : Navitrol_RequestProductionData_struct;
    SendDat : ARRAY[0..9] OF BYTE;  (* Data to send *)
    Messagesize : UINT;  (* Amount of bytes *)
    SendData : SktTCPSend;
END_VAR
VAR_INPUT
    Enable : BOOL;  (* Request to send *)
END_VAR
VAR_OUTPUT
    Done : BOOL;  (* Transmission done *)
END_VAR
VAR_INPUT
    Socket : _sSOCKET;  (* Navitrol socket *)
END_VAR
VAR_OUTPUT
    Error : BOOL;  (* Error during transmission *)
    ErrorID : WORD;  (* Error ID *)
END_VAR
VAR_INPUT
    ActivateSending : BOOL;
END_VAR
VAR
    _e1 : R_TRIG;
    _p2 : BOOL;
    _p3 : BOOL;
    _e4 : R_TRIG;
END_VAR
(* ladder, written here as Structured Text *)

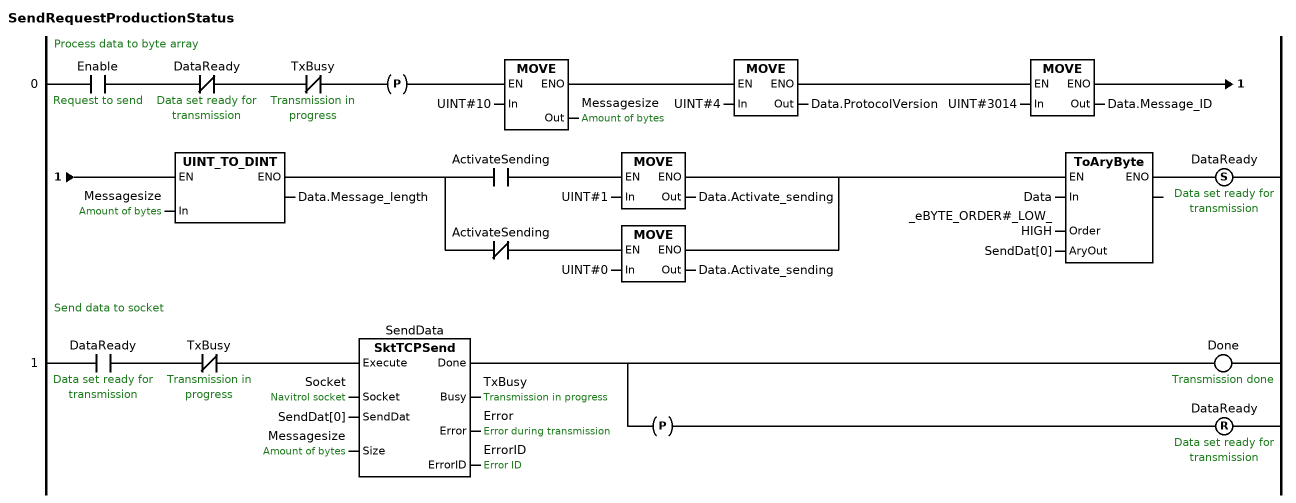
(* Rung 0: Process data to byte array *)
_e1(CLK := Enable AND NOT DataReady AND NOT TxBusy);
IF _e1.Q THEN
    Messagesize := UINT#10;
    Data.ProtocolVersion := UINT#4;
    Data.Message_ID := UINT#3014;
    Data.Message_length := UINT_TO_DINT(In := Messagesize);
END_IF;
IF _e1.Q AND ActivateSending THEN Data.Activate_sending := UINT#1; END_IF;
IF _e1.Q AND NOT ActivateSending THEN Data.Activate_sending := UINT#0; END_IF;
IF _e1.Q AND (ActivateSending OR NOT ActivateSending) THEN
    ToAryByte(In := Data, Order := _eBYTE_ORDER#_LOW_HIGH, AryOut := SendDat[0]);
    DataReady := TRUE;
END_IF;
(* Rung 1: Send data to socket *)
_p2 := DataReady AND NOT TxBusy;
SendData(Execute := _p2, Socket := Socket, SendDat := SendDat[0], Size := Messagesize, Busy => TxBusy, Error => Error, ErrorID => ErrorID);
_p3 := SendData.Done;
Done := _p3;
_e4(CLK := _p3);
IF _e4.Q THEN DataReady := FALSE; END_IF;
END_FUNCTION_BLOCK

FUNCTION_BLOCK PalletDetection_FB
VAR
    countedPallets_CTU : CTU;
    histeresisTimeForks : TON;
END_VAR
VAR_OUTPUT
    CountedPallets : INT;
END_VAR
VAR_IN_OUT
    state : Pallet_Det_State;
END_VAR
VAR_INPUT
    switchingTimeFork : TIME;
    forkSensor : BOOL;
    active : Palletdetection_Action;
    liftAtTarget : BOOL;
    liftReq : Lift_Req_State;
    liftActive : BOOL;
END_VAR
VAR_EXTERNAL
    Reset_Button : BOOL;
    MES_PalletDetection : Palletdetection_Action;
    Lift_Bot_Pos : BOOL;
END_VAR
// In init state reset counter to zero. 
IF state = init THEN 
countedPallets_CTU.Reset := TRUE;
ELSE 
countedPallets_CTU.Reset := FALSE;
END_IF;

countedPallets_CTU.PV:=10;
countedPallets_CTU(cu:=histeresisTimeForks.Q);    
histeresisTimeForks(PT:=switchingTimeFork);
if Active =Mes_NotActive THEN 
state:= init;
END_IF;

CASE State OF 
// Init state 
init:
IF Active = Mes_Active THEN 
State := assent_PLC;
END_IF;
// Pallet detection is active.
assent_PLC:
IF liftReq = Lift_Req_State#Lift_Down AND liftActive THEN 
state := lift_Goes_To_Target;
END_IF;
// Lift goes to target position.
lift_Goes_To_Target:
histeresisTimeForks(in:=forkSensor);
IF liftAtTarget THEN
state := counted_Pallets;
END_IF;
// lift is at target, 
counted_Pallets:
IF active = Mes_NotActive THEN 
state := init;
END_IF;

END_CASE;

CountedPallets := countedPallets_CTU.CV;
END_FUNCTION_BLOCK

FUNCTION_BLOCK GetCorrectedLiftHeight
VAR_INPUT
    Enable : BOOL;
    Raw_height : INT;
END_VAR
VAR_OUTPUT
    Height_INT : INT;
    Height_REAL : REAL;
END_VAR
VAR_INPUT
    Lift_height_scale : REAL;
    Lift_height_offset : INT;
END_VAR
Height_REAL := ((Raw_height * Lift_height_scale) + Lift_height_offset);
Height_INT := REAL_TO_INT(Height_REAL);
END_FUNCTION_BLOCK

FUNCTION_BLOCK LiftSpeedContoller
VAR
    V_err : REAL;
    A_scalar : REAL;
    A_set : REAL;
    Prop_Speed_Set : REAL;
    Proportional : REAL;
    Integral : REAL;
    prev_error : REAL;
    Integral_Max : REAL;
    Integral_Min : REAL;
    LiftTimeout : BOOL := False;
    Test_prop : BOOL;
END_VAR
VAR_INPUT
    Enable : BOOL;
    V_Set : REAL;  (* Velocity setpoint *)
    V_Current : REAL;  (* Current velocity *)
    V_Min : REAL;  (* Minimal velocity *)
    V_Max : REAL;  (* Maximum velocity *)
END_VAR
VAR_OUTPUT
    Prop_Speed : INT;  (* Proportional speed *)
END_VAR
VAR_INPUT
    Prop_Max_Acc : REAL;  (* Maximal proportional acceleration per cycle *)
    Prop_Speed_Max : REAL;  (* Maximal proportional speed *)
    Kp : REAL;  (* P gain *)
    Ki : REAL;  (* I gain *)
    Prop_Start_Speed : INT;  (* Start speed for controller *)
    Reset : BOOL;  (* Reset *)
    Minimal_speed_for_error : REAL;  (* Minimal speed the lift should reach before giving error *)
END_VAR
VAR_OUTPUT
    Error : BOOL;  (* Lift not moving while it should *)
    Upwards : BOOL;  (* Lift moving upwards *)
    Downwards : BOOL;  (* Lift moving downwards *)
    ActuatorActive : BOOL;  (* Actuator active *)
END_VAR
VAR_EXTERNAL
    Update_Navitrol : BOOL;
END_VAR
// Reset lift timeout when reset is true
IF Reset THEN
	LiftTimeout := FALSE;
	Error:=FALSE;
END_IF;

// Set error if lift is not moving while prop speed is maximal 
IF Prop_Speed = Prop_Speed_Max AND ABS(V_Current) < Minimal_speed_for_error THEN
	LiftTimeout := TRUE;
	Error := TRUE;
END_IF;

IF NOT Enable OR V_Set = 0 OR LiftTimeout THEN // Lift not allowed to move
	Prop_Speed := 0;
	Integral := 0; 
	Upwards := FALSE;
	Downwards := FALSE;
	ActuatorActive := FALSE;
	RETURN;
ELSIF Get10msClk() THEN // Run controller every 10ms
	
	ActuatorActive := TRUE;
	
	// Determine if lift is moving upwards or downwards
	IF V_Set > 0 THEN
		Upwards := TRUE;
		Downwards := FALSE;
	ELSIF V_Set < 0 THEN
		Upwards := FALSE;
		Downwards := TRUE;
	ELSE
		Upwards := FALSE;
		Downwards := FALSE;
	END_IF;

	// Calculate velocity error
	V_err := ABS(V_set) - ABS(V_Current);

	// Calculate the proportional and integral part
	Proportional :=  V_err * Kp;
	Integral := Integral + 0.5 * Ki * 0.01 * (V_err + prev_error) ; // 0.01 is the sample time
	
	// Provide I_gain for winding up
	IF V_Max > Proportional THEN
		Integral_Max := V_Max - Proportional;
	ELSE	
		Integral_Max := 0;
	END_IF;
	
	IF V_Min < Proportional THEN
		Integral_Min := V_Min - Proportional;
	ELSE	
		Integral_Min := 0;
	END_IF;
	
	// Clamping the integral part
	IF Integral > Integral_Max THEN
		Integral := Integral_Max;
	ELSIF Integral < Integral_Min THEN 
		Integral := Integral_Min;
	END_IF;
		
	// Calculate the A_scalar used for determine the max lift accelaration
	A_scalar := (Proportional + Integral) / V_Max; // Devided by V_max to get a value between -1 and 1
	// A_scalar := ABS(A_scalar);

	IF A_scalar > 1.0 THEN
		A_set := Prop_Max_Acc;
	ELSIF A_scalar < -1.0 THEN
		A_set := -Prop_Max_Acc;
	ELSE 
		A_set := Prop_Max_Acc * A_scalar;
	END_IF;
	
	// Calculate prop speed setpoint
	Prop_Speed_Set := Prop_Speed_Set + A_set;
	
	// Check if prop speed setpoint is within bounds
	IF Prop_Speed_Set > 0 AND Prop_Speed_Set < Prop_Speed_Max THEN
		Prop_Speed_Set := Prop_Speed_Set;
	ELSIF Prop_Speed_Set >= Prop_Speed_Max THEN 
		Prop_Speed_Set := Prop_Speed_Max;
	ELSE
		Prop_Speed_Set := 0;
	END_IF;
	
	// Set prop speed
	IF Prop_Speed = 0 AND Prop_Start_Speed > 0  THEN
		Prop_Speed :=Prop_Start_Speed;
		Prop_Speed_Set := INT_TO_REAL(Prop_Start_Speed);
	ELSE
		Prop_speed := REAL_TO_INT(Prop_Speed_Set);
	END_IF;
	
	prev_error := V_err;
	
END_IF;
END_FUNCTION_BLOCK

FUNCTION_BLOCK LiftPositionController
VAR
    H_Err : INT := 0;
    V_Scalar : REAL := 0.0;
    Kp : REAL := 0.0;
    H_set_prev : INT;
END_VAR
VAR CONSTANT
    H_MaxErr : INT := 100;
END_VAR
VAR_INPUT
    Enable : BOOL;
    H_Min : INT;  (* Minimal height *)
    H_Max : INT;  (* Maximal height *)
    V_Max : REAL;  (* Maximal velocity *)
    Kp_Up : REAL;  (* P gain for upwards movement *)
    Kp_Down : REAL;  (* P gain for downwards movement *)
    H_Set : INT := 0;  (* Height setpoint *)
    H_Current : INT;  (* Current height *)
END_VAR
VAR_OUTPUT
    At_Target : BOOL;  (* Lift at target *)
    V_Set : REAL;  (* Velocity setpoint *)
END_VAR
VAR_EXTERNAL
    ActuatorAction : BOOL;
END_VAR
IF H_set <> H_set_prev THEN
	At_target := FALSE;
	H_set_prev := H_set;
END_IF;	

// Run controller every 100 ms (10Hz)
IF Get100msClk() AND NOT At_target THEN
	
	// Calculate height error
	IF H_set >= H_min AND H_set <= H_max THEN
		H_err := H_set - H_current; 
	ELSE
		H_err := 0;
	END_IF;

	// Determine if lift has to go up or down
	IF H_err < -1 THEN
		// Lift down
		Kp := Kp_Down;
	ELSIF H_err > 1 THEN
		// Lift up
		Kp := Kp_Up; 
	ELSE
		At_target :=TRUE;
		Kp := 0.0;
		V_Set := 0;
		RETURN;
	END_IF;
	

	// Calculate velocity setpoint
	V_scalar := (INT_TO_REAL(H_err)/H_MaxErr) * Kp; 
	IF V_scalar > 1.0 THEN
		V_set := V_max;
	ELSIF V_scalar < -1.0 THEN
		V_set := -V_Max;
	ELSE
		V_set := V_max * V_scalar;
	END_IF;
	
END_IF;

IF NOT Enable THEN
	V_Set := 0;
END_IF;
END_FUNCTION_BLOCK

FUNCTION_BLOCK CalcLiftSpeed
VAR
    Index : INT := 0;
    PositionsArray : ARRAY[0..9] OF REAL;
    DeltaHeight : REAL := 0.0;
END_VAR
VAR CONSTANT
    DeltaTime : REAL := 0.01;
END_VAR
VAR
    VelocityArray : ARRAY[0..99] OF REAL;
    CurrentLiftSpeed : REAL;
    VelocitySum : REAL;
END_VAR
VAR_INPUT
    Enable : BOOL;
    CurrentLiftHeight : INT;
END_VAR
VAR_OUTPUT
    LiftSpeed : REAL;  (* Speed in m/s *)
END_VAR
// Sample each 10 ms (100HZ)
IF Get10msClk() THEN
	
	// Store last 10 measurements in array
	Index := 9;
	FOR Index := 9 TO 1 BY -1 DO
		PositionsArray[Index ] := PositionsArray[Index -1];
	END_FOR;
	PositionsArray[0] := INT_TO_REAL(CurrentLiftHeight);
	
	// Take average height difference op last 10 measurements
	DeltaHeight := PositionsArray[0] - PositionsArray[9] ;
	// CurrentLiftSpeed := (DeltaHeight / DeltaTime) ; // Speed in mm/s
	
	// Moving everage of last 10 liftspeeds
	Index := 99;
	FOR Index := 99 TO 1 BY -1 DO
		VelocityArray[Index ] := VelocityArray[Index -1];
	END_FOR;
	VelocityArray[0] := DeltaHeight;
	
	Index := 0;
	VelocitySum := 0.0;
	FOR Index := 0 TO 99 DO
		VelocitySum := VelocitySum + VelocityArray[Index];
	END_FOR;

	LiftSpeed := VelocitySum / 100 ;  // Not defided by 10 since mm/s

END_IF;
END_FUNCTION_BLOCK

FUNCTION_BLOCK ManualLift
VAR
    AutoLiftSet : BOOL;  (* Set the lift the entire action *)
    lift : BOOL;
    lift_min : BOOL;
END_VAR
VAR_INPUT
    Enable : BOOL;
    ControlMode : ControlLift;  (* Controlmode lift *)
    Button_Up : BOOL;  (* HMI button up *)
    Button_Down : BOOL;  (* HMI button down *)
    Lift_At_Target : BOOL;
    Lift_Allowed : BOOL;
    Lift_max : BOOL;
    Lift_detected_HeavyLoad : BOOL;  (* Lift has heavyload detection. *)
    Lift_height_max : INT;  (* Lift height maximum. *)
    Lift_height_min : INT;  (* Lift height minimum. *)
    Lift_height_HeavyLoad_Max : INT;  (* Lift height heavy load. *)
    Lift_Height_Actual : INT;  (* Rounded hight in mm. *)
END_VAR
VAR_IN_OUT
    Requested_Height : INT;  (* HMI requested height *)
END_VAR
VAR_OUTPUT
    Lift_Req_Manual : INT;  (* Requested height manual. *)
END_VAR
VAR_EXTERNAL
    lift_heavyLoad : BOOL;
END_VAR
VAR
    _p1 : BOOL;
    _p2 : BOOL;
    _e3 : R_TRIG;
    _e4 : F_TRIG;
    _e5 : R_TRIG;
END_VAR
(* ladder, written here as Structured Text *)

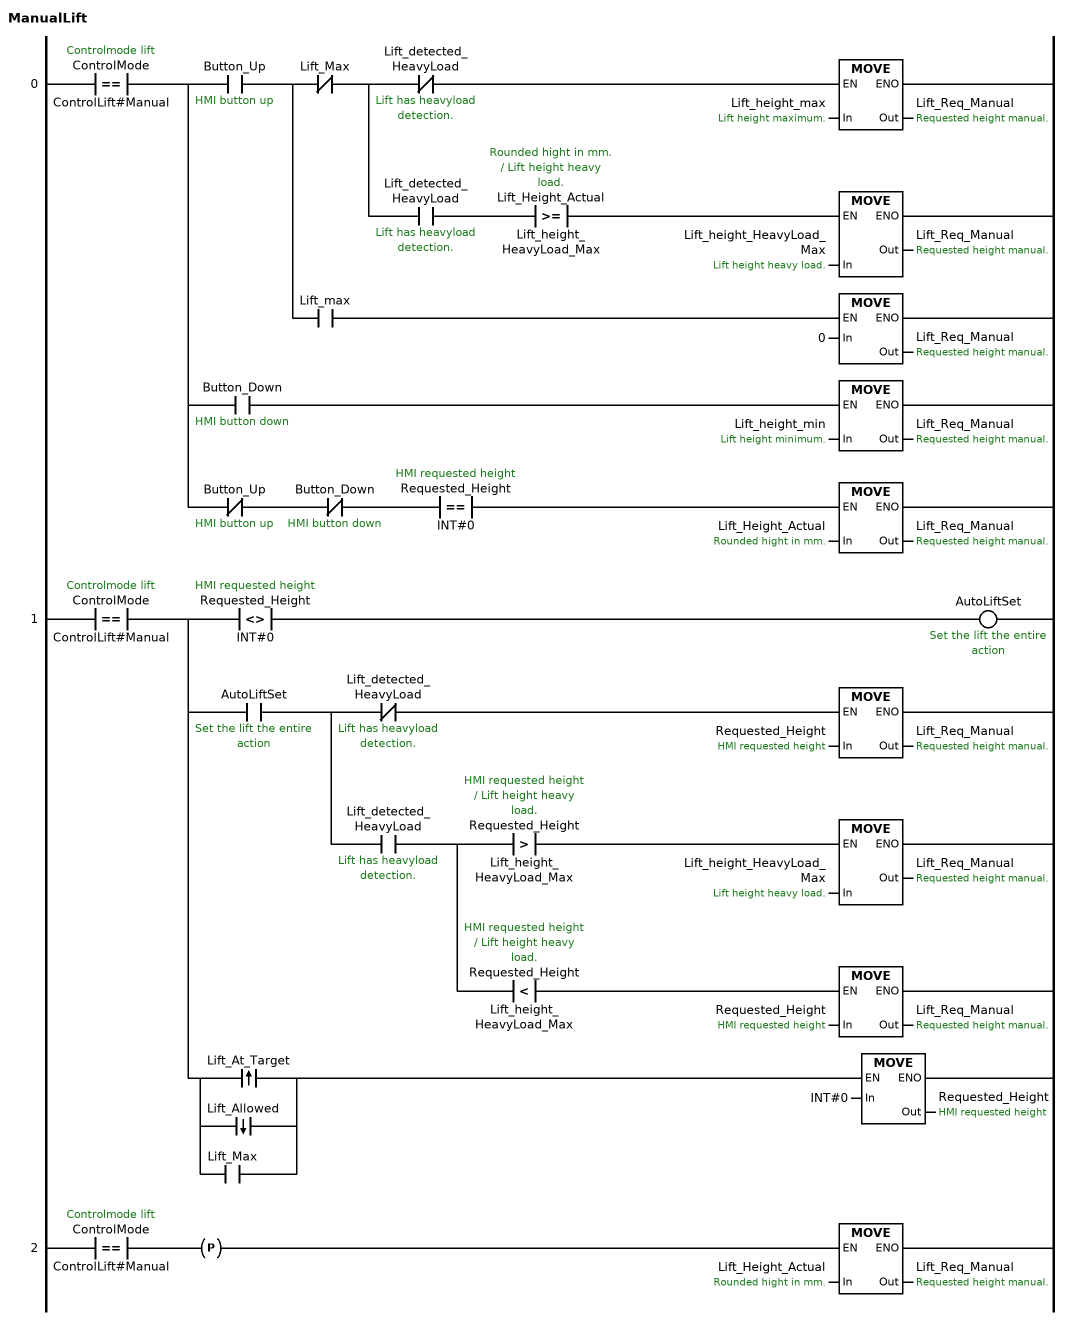
(* Rung 0 *)
_p1 := (ControlMode = ControlLift#Manual) AND Button_Up AND NOT Lift_Max;
IF _p1 AND NOT Lift_detected_HeavyLoad THEN Lift_Req_Manual := Lift_height_max; END_IF;
IF _p1 AND Lift_detected_HeavyLoad AND (Lift_Height_Actual >= Lift_height_HeavyLoad_Max) THEN
    Lift_Req_Manual := Lift_height_HeavyLoad_Max;
END_IF;
IF (ControlMode = ControlLift#Manual) AND Button_Up AND Lift_max THEN Lift_Req_Manual := 0; END_IF;
IF (ControlMode = ControlLift#Manual) AND Button_Down THEN Lift_Req_Manual := Lift_height_min; END_IF;
IF (ControlMode = ControlLift#Manual) AND NOT Button_Up AND NOT Button_Down AND (Requested_Height = INT#0) THEN
    Lift_Req_Manual := Lift_Height_Actual;
END_IF;
(* Rung 1 *)
AutoLiftSet := (ControlMode = ControlLift#Manual) AND (Requested_Height <> INT#0);
_p2 := (ControlMode = ControlLift#Manual) AND AutoLiftSet;
IF _p2 AND NOT Lift_detected_HeavyLoad THEN Lift_Req_Manual := Requested_Height; END_IF;
IF _p2 AND Lift_detected_HeavyLoad AND (Requested_Height > Lift_height_HeavyLoad_Max) THEN
    Lift_Req_Manual := Lift_height_HeavyLoad_Max;
END_IF;
IF _p2 AND Lift_detected_HeavyLoad AND (Requested_Height < Lift_height_HeavyLoad_Max) THEN
    Lift_Req_Manual := Requested_Height;
END_IF;
_e3(CLK := Lift_At_Target);
_e4(CLK := Lift_Allowed);
IF (ControlMode = ControlLift#Manual) AND (_e3.Q OR _e4.Q OR Lift_Max) THEN
    Requested_Height := INT#0;
END_IF;
(* Rung 2 *)
_e5(CLK := ControlMode = ControlLift#Manual);
IF _e5.Q THEN Lift_Req_Manual := Lift_Height_Actual; END_IF;
END_FUNCTION_BLOCK

FUNCTION_BLOCK LiftReleaseAtPosition
VAR
    x_e : REAL;
    y_e : REAL;
    MES_HeightRequest : INT;
    Lift_height_req_raw : INT;
    testINT : INT;
END_VAR
VAR_INPUT
    Enable : BOOL;
    ControlMode : ControlLift;
    Loaded : BOOL;
    Navitrol_StatusXcoord : REAL;  (* Navitrol status message X coordinate in meters *)
    Navitrol_StatusYcoord : REAL;  (* Navitrol status message Y coordinate in meters *)
    Lift_minimal_value : INT;
    Lift_maximal_value : INT;
    Lift_detected_heavyLoad : BOOL;
    Lift_height_HeavyLoad_max : INT;
    Lift_height_actual : INT;
    MES_CargoRequired : BOOL;
    MES_targetXcoord : REAL;  (* X position of MES *)
    MES_targetYcoord : REAL;  (* Y position of MES *)
    MES_TargetDistance : REAL;  (* Distance form target from inner and outer commands *)
    MES_TargetHeightInner : INT;  (* Near target actuator height *)
    MES_TargetHeightOuter : INT;  (* Far from targer actuator height *)
END_VAR
VAR_OUTPUT
    Near_Target : BOOL;  (* AGV has reached inner position *)
    MES_Lift_Req_Auto : INT;  (* Lift height request from automatic mode *)
    Near_Target_WithOut_cargo_Check : bool;
END_VAR
IF ControlMode = ControlLift#Automatic THEN
	x_e := Navitrol_StatusXcoord - (MES_targetXcoord);
	y_e := Navitrol_StatusYcoord - (MES_targetYcoord);

	Near_Target :=  (abs(x_e) < MES_TargetDistance  ) AND (abs(y_e) < MES_TargetDistance); 
	
	Near_Target_WithOut_cargo_Check := Near_Target;
	
	IF MES_CargoRequired	AND NOT loaded THEN
		Near_Target := FALSE;
	END_IF;
	
	
	IF Near_Target THEN
		MES_HeightRequest := MES_TargetHeightInner;
	ELSE
		MES_HeightRequest :=MES_TargetHeightOuter;
	END_IF;
	//check if the target height is within acceptable limits
	IF MES_HeightRequest>0 THEN 
		Lift_height_req_raw := MES_HeightRequest;
	ELSE
		Lift_height_req_raw := Lift_height_actual;
	END_IF;
	// check if there is heavy load on the forks. 
	// if this is the case, check whether the entered height is higher than heavyload. 
		IF Lift_detected_heavyLoad AND MES_HeightRequest > Lift_height_HeavyLoad_max THEN
			MES_Lift_Req_Auto :=	Lift_height_HeavyLoad_max;
		ELSE	
		IF (Lift_height_req_raw <  Lift_minimal_value) THEN
			MES_Lift_Req_Auto := Lift_minimal_value;
		ELSIF (Lift_height_req_raw > Lift_maximal_value) THEN
			MES_Lift_Req_Auto := Lift_maximal_value;
		ELSE
		MES_Lift_Req_Auto := Lift_height_req_raw;	
		END_IF;
	END_IF;
END_IF;
END_FUNCTION_BLOCK

FUNCTION_BLOCK LiftLoadStatus
VAR_INPUT
    Enable : BOOL;  (* AGV uses an analog sensor for load detection *)
    Analog_load : BOOL;
    Load1 : BOOL;  (* Load sensor 1 *)
    Load2 : BOOL;  (* Load sensor 2 *)
    Load_Distance : real;  (* Distance to load *)
    AnalogLoad_Cargo_Max : REAL;  (* Valid cargo range *)
    AnalogLoad_Min : REAL;  (* Minimum value for cargo on fork *)
    AnalogLoad_Max : REAL;  (* Fork distance for fork *)
    Near_Target : BOOL;  (* AGV has reached inner position *)
    Lift_Move_Up : BOOL;  (* lift is moving up *)
END_VAR
VAR_OUTPUT
    Cargo_Ok : BOOL;  (* Cargo_Ok *)
    AGV_AtCargo : BOOL;  (* AGV has reached the cargo *)
    ForkBlocked : BOOL;  (* Analog sensor detects object on fork *)
    Agv_Loaded : BOOL;
END_VAR
VAR_INPUT
    Lift_Move_down : BOOL;
END_VAR
VAR_EXTERNAL
    AnalogLoad : BOOL;
    AgvLoaded : BOOL;
END_VAR
VAR
    _e1 : R_TRIG;
    _e2 : F_TRIG;
    _p3 : BOOL;
END_VAR
(* ladder, written here as Structured Text *)

